// TIA Portal V19 program export: 3 tag tables, 4 data types, 23 data blocks, 30 code blocks (in call order from the OBs), 38 instance data blocks

VAR_GLOBAL   // PLC tag table "Safety_IO"
   IS_EstopLeftRopePull AT %I500.1 : Bool;   // Right e-stop rope pull switch - Channel 1   {ExternalAccessible false}
   IS_EstopRightRopePull AT %I500.0 : Bool;   // Left e-stop rope pull switch - Channel 1   {ExternalAccessible false}
   IS_EStopMainCabinet AT %I500.2 : Bool;   // Main panel e-stop - Channel 1   {ExternalAccessible false}
   IS_EStopEntryDoor AT %I500.3 : Bool;   // Entry door e-stop - Channel 1   {ExternalAccessible false}
   IS_EstopLeftRopePull_Ch2 AT %I500.5 : Bool;   // Right e-stop rope pull switch - Channel 2   {ExternalAccessible false}
   IS_EstopRightRopePull_Ch2 AT %I500.4 : Bool;   // Left e-stop rope pull switch - Channel 2   {ExternalAccessible false}
   IS_EStopMainCabinet_Ch2 AT %I500.6 : Bool;   // Main panel e-stop - Channel 2   {ExternalAccessible false}
   IS_EStopEntryDoor_Ch2 AT %I500.7 : Bool;   // Entry door e-stop - Channel 2   {ExternalAccessible false}
   IS_DoorAcces_Ch1 AT %I507.0 : Bool;   // Door acces state - Channel 1   {ExternalAccessible false}
   IS_GateAccesCBS AT %I507.1 : Bool;   // CBS Gate Acces State - Channel 1   {ExternalAccessible false}
   IS_EStopControlRoom AT %I507.2 : Bool;   // Control Room E-Stop - Channel 1   {ExternalAccessible false}
   IS_DoorAcces_Ch2 AT %I507.4 : Bool;   // Door acces state - Channel 2   {ExternalAccessible false}
   IS_GateAccesCBS_Ch2 AT %I507.5 : Bool;   // CBS Gate Acces State - Channel 2   {ExternalAccessible false}
   IS_EStopControlRoom_Ch2 AT %I507.6 : Bool;   // Control Room E-Stop - Channel 2   {ExternalAccessible false}
   OS_EStopSuctionUnit AT %Q522.1 : Bool;   // E-Stop Suction Unit   {ExternalAccessible false}
   OS_EnableAirSupplyLeftRobot AT %Q522.2 : Bool;   // Air supply robot 1 Ok   {ExternalAccessible false}
   OS_EnableAirSupplyRightRobot AT %Q522.3 : Bool;   // Air supply robot 2 Ok   {ExternalAccessible false}
   OS_EnableAirSupplySuctionUnit AT %Q522.4 : Bool;   // Air supply suction unit Ok   {ExternalAccessible false}
   ISS_EStopSuctionUnit AT %I522.1 : Bool;   // State E-Stop Suction Unit   {ExternalAccessible false}
   ISS_EnableAirSupplyLeftRobot AT %I522.2 : Bool;   // State Air supply robot 1 Ok   {ExternalAccessible false}
   ISS_EnableAirSupplyRightRobot AT %I522.3 : Bool;   // State Air supply robot 2 Ok   {ExternalAccessible false}
   ISS_EnableAirSupplySuctionUnit AT %I522.4 : Bool;   // Air supply suction unit Ok   {ExternalAccessible false}
   ISS_EstopLeftRopePull AT %I501.1 : Bool;   // State Right e-stop rope pull switch - Channel 1   {ExternalAccessible false}
   ISS_EstopRightRopePull AT %I501.0 : Bool;   // State Left e-stop rope pull switch - Channel 1   {ExternalAccessible false}
   ISS_EStopMainCabinet AT %I501.2 : Bool;   // State Main panel e-stop - Channel 1   {ExternalAccessible false}
   ISS_EStopEntryDoor AT %I501.3 : Bool;   // State Entry door e-stop - Channel 1   {ExternalAccessible false}
   ISS_DoorAcces_Ch1 AT %I508.0 : Bool;   // State Door acces state - Channel 1   {ExternalAccessible false}
   ISS_GateAccesCBS AT %I508.1 : Bool;   // State CBS Gate Acces State - Channel 1   {ExternalAccessible false}
   ISS_EStopControlRoom AT %I508.2 : Bool;   // State Control Room E-Stop - Channel 1   {ExternalAccessible false}
   ISS_DoorAcces_Ch2 AT %I508.4 : Bool;   // State Door acces state - Channel 2   {ExternalAccessible false}
   ISB_500 AT %IB500 : SInt;   //    {ExternalWritable false}
   ISB_507 AT %IB507 : SInt;   //    {ExternalWritable false}
   ISB_514 AT %IB514 : SInt;   //    {ExternalWritable false}
   OSB_522 AT %QB522 : SInt;   //    {ExternalWritable false}
   IS_PedestrialDoor AT %I507.3 : Bool;   // Pedestral door acces control   {ExternalAccessible false}
   IS_CaptiveKeyState AT %I514.0 : Bool;   // Captive key in lock - Channel 1   {ExternalAccessible false}
   IS_CaptiveKeyState_Ch2 AT %I514.4 : Bool;   // Captive key in lock - Channel 2   {ExternalAccessible false}
   ISS_CaptiveKeyState AT %I515.0 : Bool;   // State Captive key in lock   {ExternalAccessible false}
   IS_VacuumPumpRunning AT %I507.7 : Bool;   // Vacuum pump runing, zero speed detection   {ExternalAccessible false}
END_VAR

VAR_GLOBAL   // PLC tag table "Standard_IO"
   I_IPBDoorAccesRequest AT %I100.0 : Bool;   // Illuminate push button acces request   {ExternalAccessible false}
   I_IPBCloseDoor AT %I100.1 : Bool;   // Illuminate push button close door   {ExternalAccessible false}
   I_EStopState AT %I100.2 : Bool;   // Entry door AU state   {ExternalAccessible false}
   I_DoorClosed AT %I100.3 : Bool;   // Entry door state 1   {ExternalAccessible false}
   I_BoltTongueInserted AT %I100.4 : Bool;   // Entry door state 2   {ExternalAccessible false}
   I_GuardLocked AT %I100.5 : Bool;   // Entry door state 3   {ExternalAccessible false}
   I_FaultPresent AT %I100.6 : Bool;   // Entry door state 4   {ExternalAccessible false}
   I_PSAirLeftRobotOk AT %I101.0 : Bool;   // Air supply robot 1 Ok   {ExternalAccessible false}
   I_PSAirRightRobotOk AT %I101.1 : Bool;   // Air supply robot 2 Ok   {ExternalAccessible false}
   I_PSAirSuctionUnitOk AT %I101.2 : Bool;   // Air supply suction unit Ok   {ExternalAccessible false}
   I_FanDriveRunning AT %I101.4 : Bool;   // Suction unit - Fan Drive Running   {ExternalAccessible false}
   I_DustBagFull AT %I101.5 : Bool;   // Suction unit - Dust bag full   {ExternalAccessible false}
   I_FanDriveFault AT %I101.6 : Bool;   // Suction unit - Fan Drive fault   {ExternalAccessible false}
   I_SequencerFault AT %I101.7 : Bool;   // Suction unit - Sequencer in fault   {ExternalAccessible false}
   O_IPBDoorAccesRequest AT %Q100.0 : Bool;   // Illuminate push button acces request   {ExternalAccessible false}
   O_IPBCloseDoor AT %Q100.1 : Bool;   // Illuminate push button close door   {ExternalAccessible false}
   O_ResetDoorFault AT %Q100.2 : Bool;   // Reset fault on door   {ExternalAccessible false}
   O_SignalToweGreenLight AT %Q100.4 : Bool;   // Light towers - green light   {ExternalAccessible false}
   O_SignalToweOrangeLight AT %Q100.5 : Bool;   // Light towers - orange light   {ExternalAccessible false}
   O_SignalToweRedLight AT %Q100.6 : Bool;   // Light towers - red light   {ExternalAccessible false}
   O_SignalToweHorn AT %Q100.7 : Bool;   // Light towers - horn   {ExternalAccessible false}
   O_StartVacuum AT %Q101.4 : Bool;   // Suction unit - Vacuum On   {ExternalAccessible false}
   O_StopVacuum AT %Q101.5 : Bool;   // Suction unit - Vacuum Off   {ExternalAccessible false}
   O_TeepTrackCycleTimeR1 AT %Q102.0 : Bool;   // Alstom Teep track Cycle Time Robot 1 (Left)   {ExternalAccessible false}
   O_TeepTrackStartStopR1 AT %Q102.1 : Bool;   // Alstom Teep track Start and Stop Robot 1 (Left)   {ExternalAccessible false}
   O_LockDoor AT %Q101.0 : Bool;   // Lock acces door   {ExternalAccessible false}
   OST_SendLeft AT %Q106.0 : "stMasterToSlave";   // Send information to left slave PLC   {ExternalAccessible false}
   OST_SendRight AT %Q234.0 : "stMasterToSlave";   // Send information to right slave PLC   {ExternalAccessible false}
   IST_ReceiveLeft AT %I106.0 : "stSlaveToMaster";   // Receive information from left slave PLC   {ExternalAccessible false}
   IST_ReceiveRight AT %I234.0 : "stSlaveToMaster";   // Receive information from right slave PLC   {ExternalAccessible false}
   I_FanFault AT %I102.0 : Bool;   // Suction unit - Fan fault   {ExternalAccessible false}
   I_ValveMotorFault AT %I102.1 : Bool;   // Suction unit - Valve Motor Fault   {ExternalAccessible false}
   IB_100 AT %IB100 : SInt;   //    {ExternalWritable false}
   IB_101 AT %IB101 : SInt;   //    {ExternalWritable false}
   IB_102 AT %IB102 : SInt;   //    {ExternalWritable false}
   IB_103 AT %IB103 : SInt;   //    {ExternalWritable false}
   OB_100 AT %QB100 : SInt;   //    {ExternalWritable false}
   OB_101 AT %QB101 : SInt;   //    {ExternalWritable false}
   OB_102 AT %QB102 : SInt;   //    {ExternalWritable false}
   OB_103 AT %QB103 : SInt;   //    {ExternalWritable false}
   O_TeepTrackCycleTimeR2 AT %Q102.2 : Bool;   // Alstom Teep track Cycle Time Robot 2 (Right)   {ExternalAccessible false}
   O_TeepTrackStartStopR2 AT %Q102.3 : Bool;   // Alstom Teep track Start and Stop Robot 2 (Right)   {ExternalAccessible false}
END_VAR

VAR_GLOBAL   // PLC tag table "System"
   System_Byte AT %MB1 : Byte;
   FirstScan AT %M1.0 : Bool;
   DiagStatusUpdate AT %M1.1 : Bool;
   AlwaysTRUE AT %M1.2 : Bool;
   AlwaysFALSE AT %M1.3 : Bool;
   Clock_Byte AT %MB0 : Byte;
   Clock_10Hz AT %M0.0 : Bool;
   Clock_5Hz AT %M0.1 : Bool;
   "Clock_2.5Hz" AT %M0.2 : Bool;
   Clock_2Hz AT %M0.3 : Bool;
   "Clock_1.25Hz" AT %M0.4 : Bool;
   Clock_1Hz AT %M0.5 : Bool;
   "Clock_0.625Hz" AT %M0.6 : Bool;
   "Clock_0.5Hz" AT %M0.7 : Bool;
   ShuntTempSeb AT %M10.0 : Bool;
   ISS_PedestrialDoor AT %I508.3 : Bool;   // State Pedestral door acces control
   ISS_VacuumPumpRunning AT %I508.7 : Bool;   // State Vacuum pump runing, zero speed detection
END_VAR

TYPE "stConfigGrease"
   STRUCT
      uiNbPulsePerKm : UInt := 4411;   // Number of pulse per km
      uiKmForGreasing : UInt := 32;   // Number of Km between each greasing
      tTimeEnableGreasePump : Time := T#1M;   // Time of enabling grease pump
      tTimeoutPxGrease : Time := T#1M;   // Timeout for the proxy greas
   END_STRUCT;
END_TYPE

TYPE "stFlatnessData"
   STRUCT
      xFlatnessCrtlRequestRecord { ExternalAccessible := 'False'; ExternalVisible := 'False'; ExternalWritable := 'False'} : Bool;
      xFlatnessCtrlRecorded { ExternalAccessible := 'False'; ExternalVisible := 'False'; ExternalWritable := 'False'} : Bool;
      xFlatnessCtrlPassed { ExternalAccessible := 'False'; ExternalVisible := 'False'; ExternalWritable := 'False'} : Bool;
      uiStrokePositionDiskA { ExternalAccessible := 'False'; ExternalVisible := 'False'; ExternalWritable := 'False'} : UInt;
      uiStrokePositionDiskB { ExternalAccessible := 'False'; ExternalVisible := 'False'; ExternalWritable := 'False'} : UInt;
      uiStrokePositionDiskC { ExternalAccessible := 'False'; ExternalVisible := 'False'; ExternalWritable := 'False'} : UInt;
   END_STRUCT;
END_TYPE

TYPE "stItemListRecipe"
   STRUCT
      RecipeName { ExternalAccessible := 'False'; ExternalVisible := 'False'; ExternalWritable := 'False'} : String[30];
      RecipeIndex { ExternalAccessible := 'False'; ExternalVisible := 'False'; ExternalWritable := 'False'} : USInt;
   END_STRUCT;
END_TYPE

TYPE "stParamManuFerRobotic"
   STRUCT
      "#OutToSlave.ManualSandingPaperParam.nSetForceTarget    #OutToSlave.ManualSandingPaperParam.nSetForceZero    #OutToSlave.ManualSa" : Bool;
   END_STRUCT;
END_TYPE

DATA_BLOCK "DB_CurrentRecipe"   // DB5
{ S7_Optimized_Access := 'TRUE'; DB_Accessible_From_OPC_UA := 'FALSE' }
// stored: AutoNumber false, DBAccessibleFromOPCUA false, DBAccessibleFromWebserver false, MemoryReserve 100
   VAR RETAIN
      usiCurrentRecipeNumber : USInt;
      usiCurrentLayerType : USInt;
      usiCurrentJobDataLeft { ExternalAccessible := 'False'; ExternalVisible := 'False'; ExternalWritable := 'False'} : USInt;
      usiCurrentJobDataRight { ExternalAccessible := 'False'; ExternalVisible := 'False'; ExternalWritable := 'False'} : USInt;
      uiCdbNumber : UInt;
      CompleteRecipe : "stRecipe";
      WorkRecipe { S7_SetPoint := 'True'} : "stWorkRecipe";
   END_VAR
BEGIN
END_DATA_BLOCK

DATA_BLOCK "DB_Exchange"   // DB1
{ S7_Optimized_Access := 'TRUE'; DB_Accessible_From_OPC_UA := 'FALSE' }
// stored: AutoNumber false, DBAccessibleFromOPCUA false, DBAccessibleFromWebserver false, MemoryReserve 100
   VAR
      xAutoMode { ExternalAccessible := 'False'; ExternalVisible := 'False'; ExternalWritable := 'False'} : Bool;   // Automatic mode
      xSemiAutoMode { ExternalAccessible := 'False'; ExternalVisible := 'False'; ExternalWritable := 'False'} : Bool;   // Semi-automatic mode
      xMaintenanceMode { ExternalAccessible := 'False'; ExternalVisible := 'False'; ExternalWritable := 'False'} : Bool;   // Maintenance mode
      xAuthorizationStartSanding { ExternalAccessible := 'False'; ExternalVisible := 'False'; ExternalWritable := 'False'} : Bool;
      xLeftRobotStartVacuum { ExternalAccessible := 'False'; ExternalVisible := 'False'; ExternalWritable := 'False'} : Bool;   // Left Robot request start vacuum
      xRightRobotStartVacuum { ExternalAccessible := 'False'; ExternalVisible := 'False'; ExternalWritable := 'False'} : Bool;   // Right Robot request start vacuum
      xStopRobotRequested { ExternalAccessible := 'False'; ExternalVisible := 'False'; ExternalWritable := 'False'} : Bool;   // Stop robot requested for openning the door
      xLeftRobotStopped { ExternalAccessible := 'False'; ExternalVisible := 'False'; ExternalWritable := 'False'} : Bool;   // Left Robot stopped in good position
      xRightRobotStopped { ExternalAccessible := 'False'; ExternalVisible := 'False'; ExternalWritable := 'False'} : Bool;   // Right Robot stopped in good position
      xGlobalFault { ExternalAccessible := 'False'; ExternalVisible := 'False'; ExternalWritable := 'False'} : Bool;   // Cell Global Fault
      xGlobalWarning { ExternalAccessible := 'False'; ExternalVisible := 'False'; ExternalWritable := 'False'} : Bool;   // Cell Global warning
      xInformation { ExternalAccessible := 'False'; ExternalVisible := 'False'; ExternalWritable := 'False'} : Bool;   // An information message is display
      xConditionOk { ExternalAccessible := 'False'; ExternalVisible := 'False'; ExternalWritable := 'False'} : Bool;   // Condition to run ok
      xStartUpWarningLeft { ExternalAccessible := 'False'; ExternalVisible := 'False'; ExternalWritable := 'False'} : Bool;   // Start up warning before left robot run
      xStartUpWarningRight { ExternalAccessible := 'False'; ExternalVisible := 'False'; ExternalWritable := 'False'} : Bool;   // Start up warning before right robot run
      xReqOperatorAction { ExternalAccessible := 'False'; ExternalVisible := 'False'; ExternalWritable := 'False'} : Bool;   // Request operator action
      xRecipeOpeInProgress { ExternalAccessible := 'False'; ExternalVisible := 'False'; ExternalWritable := 'False'} : Bool;   // Recipe Operation in progress
      xSandingInProgress { ExternalAccessible := 'False'; ExternalVisible := 'False'; ExternalWritable := 'False'} : Bool;   // Sanding process is in progress
      xUnloadRecipe { ExternalAccessible := 'False'; ExternalVisible := 'False'; ExternalWritable := 'False'} : Bool;   // Unload current recipe
      xProductionRunningRobot1 { ExternalAccessible := 'False'; ExternalVisible := 'False'; ExternalWritable := 'False'} : Bool;   // Production running on Robot 1
      xProductionRunningRobot2 { ExternalAccessible := 'False'; ExternalVisible := 'False'; ExternalWritable := 'False'} : Bool;   // Production running on Robot 2
      xStartSanding { ExternalAccessible := 'False'; ExternalVisible := 'False'; ExternalWritable := 'False'} : Bool;   // Beginning of sanding
      xEndSanding { ExternalAccessible := 'False'; ExternalVisible := 'False'; ExternalWritable := 'False'} : Bool;   // End of sanding
      udiVacuumRunningTime { ExternalAccessible := 'False'; ExternalVisible := 'False'; ExternalWritable := 'False'} : UDInt;   // Vacuum Running time
      LeftRobot { ExternalAccessible := 'False'; ExternalVisible := 'False'; ExternalWritable := 'False'} : Struct
         udiFaultTime : UDInt;
         udiRunTime : UDInt;
         udiPauseTime : UDInt;
         udiRobotPowerOnTime : UDInt;
         udiRobotDriveOnTime : UDInt;
         xRobotUsed : Bool;
      END_STRUCT;
      RightRobot { ExternalAccessible := 'False'; ExternalVisible := 'False'; ExternalWritable := 'False'} : Struct
         udiFaultTime : UDInt;
         udiRunTime : UDInt;
         udiPauseTime : UDInt;
         udiRobotPowerOnTime : UDInt;
         udiRobotDriveOnTime : UDInt;
         xRobotUsed : Bool;
      END_STRUCT;
      stLeftRobotFlatnessCtrlData { ExternalAccessible := 'False'; ExternalVisible := 'False'; ExternalWritable := 'False'} : "stFlatnessData";
      stRightRobotFlatnessCtrlData { ExternalAccessible := 'False'; ExternalVisible := 'False'; ExternalWritable := 'False'} : "stFlatnessData";
   END_VAR
BEGIN
END_DATA_BLOCK

DATA_BLOCK "DB_JobData"   // DB3
{ S7_Optimized_Access := 'TRUE'; DB_Accessible_From_OPC_UA := 'FALSE' }
// stored: AutoNumber false, DBAccessibleFromOPCUA false, DBAccessibleFromWebserver false, MemoryReserve 100
   VAR RETAIN
      aJobData : Array[0..99] of "stJobData";   // Array of job data parameters
   END_VAR
BEGIN
END_DATA_BLOCK

DATA_BLOCK "DB_Parameters"   // DB2
{ S7_Optimized_Access := 'TRUE'; DB_Accessible_From_OPC_UA := 'FALSE' }
// stored: DBAccessibleFromOPCUA false, DBAccessibleFromWebserver false, MemoryReserve 100
   VAR RETAIN
      CommMainPanel { ExternalAccessible := 'False'; ExternalVisible := 'False'; ExternalWritable := 'False'} : TCON_IP_v4;
      CommLeftRobot { ExternalAccessible := 'False'; ExternalVisible := 'False'; ExternalWritable := 'False'} : TCON_IP_v4;
      CommRightRobot { ExternalAccessible := 'False'; ExternalVisible := 'False'; ExternalWritable := 'False'} : TCON_IP_v4;
      tDelatBetweenReady { ExternalAccessible := 'False'; ExternalVisible := 'False'; ExternalWritable := 'False'} : Time := T#1s;
   END_VAR
BEGIN
   CommMainPanel.InterfaceId := 64;
   CommMainPanel.ID := 16#01;
   CommMainPanel.ConnectionType := 16#0B;
   CommMainPanel.ActiveEstablished := TRUE;
   CommMainPanel.RemoteAddress.ADDR[1] := 192;
   CommMainPanel.RemoteAddress.ADDR[2] := 168;
   CommMainPanel.RemoteAddress.ADDR[3] := 1;
   CommMainPanel.RemoteAddress.ADDR[4] := 20;
   CommMainPanel.RemotePort := 502;
   CommLeftRobot.InterfaceId := 64;
   CommLeftRobot.ID := 16#02;
   CommLeftRobot.ConnectionType := 16#0B;
   CommLeftRobot.ActiveEstablished := TRUE;
   CommLeftRobot.RemoteAddress.ADDR[1] := 192;
   CommLeftRobot.RemoteAddress.ADDR[2] := 168;
   CommLeftRobot.RemoteAddress.ADDR[3] := 1;
   CommLeftRobot.RemoteAddress.ADDR[4] := 21;
   CommLeftRobot.RemotePort := 502;
   CommRightRobot.InterfaceId := 64;
   CommRightRobot.ID := 16#03;
   CommRightRobot.ConnectionType := 16#0B;
   CommRightRobot.ActiveEstablished := TRUE;
   CommRightRobot.RemoteAddress.ADDR[1] := 192;
   CommRightRobot.RemoteAddress.ADDR[2] := 168;
   CommRightRobot.RemoteAddress.ADDR[3] := 1;
   CommRightRobot.RemoteAddress.ADDR[4] := 22;
   CommRightRobot.RemotePort := 503;
END_DATA_BLOCK

DATA_BLOCK "DB_FromHmi"   // DB29
{ S7_Optimized_Access := 'TRUE'; DB_Accessible_From_OPC_UA := 'FALSE' }
// stored: AutoNumber false, DBAccessibleFromOPCUA false, DBAccessibleFromWebserver false, MemoryReserve 100
   VAR
      xLightTest : Bool;   // Light test
      xResetFault : Bool;   // Reset fault and safety
      xStartVacuum : Bool;   // Start vacuum
      xStopVacuum : Bool;   // Stop vacuum
      xReqChangeBigbag : Bool;   // Request change Bigbag
      xValidationBigbagChanged : Bool;   // Validation operator bigbag changed
      xListRecipe : Bool;   // Do the list of all the recipe available in the data base
      xLoadRecipe : Bool;   // Load current recipe from data base
      xSaveRecipe : Bool;   // Save current recipe into the data base
      xNewRecipe : Bool;   // Select next free recipe on the data base
      xDeleteRecipe : Bool;   // Delete the recipe from the data base
      xNextRecipe : Bool;   // Load next recipe in the data base
      xPrevRecipe : Bool;   // Load previus recipe in the data base
      xValideOperation : Bool;   // Validation Operator to remove or Put disk on FerRobotic head
      xValideFault : Bool;   // Validation Operator of Flatness fault
      xProdRecordNext : Bool;
      xProdRecordPrev : Bool;
      xProdRecordDeleteAll : Bool;
      xFlatRecNextLeftRobot : Bool;
      xFlatRecPrevLeftRobot : Bool;
      xFlatRecDelAllLeftRobot : Bool;
      xFlatRecNextRightRobot : Bool;
      xFlatRecPrevRightRobot : Bool;
      xFlatRecDelAllRightRobot : Bool;
   END_VAR
   VAR RETAIN
      xEnableStartLeftRobot : Bool;   // Enable start robot
      xEnableStartRightRobot : Bool;   // Enable start robot
   END_VAR
   VAR
      xDryRun : Bool;   // Robot run in DryRun
      xExportProdData : Bool;
      xExportFlatCtrlRobot1 : Bool;
      xExportFlatCtrlRobot2 : Bool;
      uiCurentRecord : UInt;
      uiFlatCurentRecLeftRobot : UInt;
      uiFlatCurentRecRightRobot : UInt;
      uiDisplayJobNumber : UInt;
   END_VAR
   VAR RETAIN
      usiOperatingMode : USInt;   // Operating mode (1 = Semi-Auto, 2 = Auto)
      uiUserGroup : USInt;   // User grope number logged on HMI
   END_VAR
   VAR
      LeftRobot : Struct   // Command for left robot
         xResetGrafcet : Bool;   // Reset robot communication grafcet
         xStartCycle : Bool;   // Start Cycle
         xStopCycle : Bool;   // Stop Cycle
         xCancelCycle : Bool;   // Cancel cycle
         xStopEndCycle : Bool;   // Stop end of cycle
         xReqChangeDisk : Bool;
         xStartServicePath : Bool;   // Start service path
         xStopServicePath : Bool;   // Stop service path
         xCancelServicePath : Bool;   // Cancel service path
         usiJobNumberDisplay : USInt;   // Job number displayed for robot left
         uiServicePathNumber : UInt;   // Service path number
         xCmdManuLockGimball : Bool;
         xCmdManuLockEccentric1 : Bool;
         xCmdManuLockEccentric2 : Bool;
         xCmdManuLockEccentric3 : Bool;
         xCmdManuEnableRotate : Bool;
         xCmdManuCloseVacValve : Bool;
         xCmdManuOpenVacValve : Bool;
         xCmdManuRemoveConfig : Bool;   // Manual command for activate the Remove config on FerRobotic Head
         xCmdManuPickupConfig : Bool;   // Manual command for activate the Pickup config on FerRobotic Head
         xCmdManuFlatnessConfig : Bool;   // Manual command for activate the Flatness check config on FerRobotic Head
         xMaintStartProg : Bool;
         xMaintStartMain : Bool;
         xForceLubricationX : Bool;
         xForceLubricationZ : Bool;
         ParamManu : "stFerRoboticParam";
      END_STRUCT;
      RightRobot : Struct   // Commande for right robot
         xResetGrafcet : Bool;   // Reset robot communication grafcet
         xStartCycle : Bool;   // Start Cycle
         xStopCycle : Bool;   // Stop Cycle
         xCancelCycle : Bool;   // Cancel cycle
         xStopEndCycle : Bool;   // Stop end of cycle
         xReqChangeDisk : Bool;
         xStartServicePath : Bool;   // Start service path
         xStopServicePath : Bool;   // Stop service path
         xCancelServicePath : Bool;   // Cancel service path
         usiJobNumberDisplay : USInt;   // Job number displayed for robot right
         uiServicePathNumber : UInt;   // Service path number
         xCmdManuLockGimball : Bool;
         xCmdManuLockEccentric1 : Bool;
         xCmdManuLockEccentric2 : Bool;
         xCmdManuLockEccentric3 : Bool;
         xCmdManuEnableRotate : Bool;
         xCmdManuCloseVacValve : Bool;
         xCmdManuOpenVacValve : Bool;
         xCmdManuRemoveConfig : Bool;   // Manual command for activate the Remove config on FerRobotic Head
         xCmdManuPickupConfig : Bool;   // Manual command for activate the Pickup config on FerRobotic Head
         xCmdManuFlatnessConfig : Bool;   // Manual command for activate the Flatness check config on FerRobotic Head
         xMaintStartProg : Bool;
         xMaintStartMain : Bool;
         xForceLubricationX : Bool;
         xForceLubricationZ : Bool;
         ParamManu : "stFerRoboticParam";
      END_STRUCT;
   END_VAR
BEGIN
END_DATA_BLOCK

DATA_BLOCK "DB_HmiLight"   // DB27
{ S7_Optimized_Access := 'TRUE' }
// stored: AutoNumber false, MemoryReserve 100
   VAR
      xMemFpClock { ExternalAccessible := 'False'; ExternalVisible := 'False'; ExternalWritable := 'False'} : Bool;
      xFpClock { ExternalAccessible := 'False'; ExternalVisible := 'False'; ExternalWritable := 'False'} : Bool;
   END_VAR
BEGIN
END_DATA_BLOCK

DATA_BLOCK "DB_PointerHMI"   // DB25
{ S7_Optimized_Access := 'TRUE'; DB_Accessible_From_OPC_UA := 'FALSE' }
// stored: AutoNumber false, DBAccessibleFromOPCUA false, DBAccessibleFromWebserver false, MemoryReserve 100
   VAR
      Coordination : Word;
      ProjectID : Word;
      ScreenNumber : Array[0..4] of Word;
      JobMailbox : Array[0..3] of Word;
   END_VAR
BEGIN
END_DATA_BLOCK

DATA_BLOCK "DB_ToHmi"   // DB28
{ S7_Optimized_Access := 'TRUE'; DB_Accessible_From_OPC_UA := 'FALSE' }
// stored: AutoNumber false, DBAccessibleFromOPCUA false, DBAccessibleFromWebserver false, MemoryReserve 100
   VAR
      xShowPopReqChangeBigbag : Bool;   // Show Popup change Bigbag requested
      xShowPopNoMoreRecipeAvailable : Bool;   // Show Popup no more recipe available in the data base
      xSafetyState { ExternalWritable := 'False'} : Bool;   // Safety State
      xDiseableRecipeButton { ExternalWritable := 'False'} : Bool;   // Diseable all button for manage recipe
      xDisplayPrevButton { ExternalWritable := 'False'} : Bool;   // Display previous button in recipe screen
      xDisplayNextButton { ExternalWritable := 'False'} : Bool;   // Display next button in recipe screen
      xDiseableNewButton { ExternalWritable := 'False'} : Bool;   // Diseable new recipe button
      xDiseableSaveButton { ExternalWritable := 'False'} : Bool;   // Diseable save recipe button
      xDiseableDeleteButton { ExternalWritable := 'False'} : Bool;   // Diseable delete recipe button
      xLockRecipe { ExternalWritable := 'False'} : Bool;   // Lock recipe during production
      xLockSelectJobDataNumber { ExternalWritable := 'False'} : Bool;   // Lock selection of job data number
      xLockJobDataLeft { ExternalWritable := 'False'} : Bool;   // Lock modification Job Data left robot
      xLockJobDataRight { ExternalWritable := 'False'} : Bool;   // Lock modification Job Data right robot
      xVacuumPumpRunning { ExternalWritable := 'False'} : Bool;
      xVacuumDriveActivated { ExternalWritable := 'False'} : Bool;
      xLockMaintenance { ExternalWritable := 'False'} : Bool;   // Lock button to switch in Maintenance mode
      xLockSemiAuto { ExternalWritable := 'False'} : Bool;   // Lock button to switch in Semi-Auto mode
      xHomePositionR1 { ExternalWritable := 'False'} : Bool;   // Robot 1 in Home Position
      xHomePositionR2 { ExternalWritable := 'False'} : Bool;   // Robot 2 in Home Position
      xAccessDoor { ExternalWritable := 'False'} : Bool;   // Access door closed
      xCaptiveKey { ExternalWritable := 'False'} : Bool;   // Captive key on contact switch
      xLightBeam { ExternalWritable := 'False'} : Bool;   // Light Beam clear
      xCbsGate { ExternalWritable := 'False'} : Bool;   // CBS Gate closed
      nGlobalState { ExternalWritable := 'False'} : Int;   // Cell global state
      wVacuumState { ExternalWritable := 'False'} : Word;
      uiProdRecordMin { ExternalWritable := 'False'} : UInt;   // Mini record number
      uiProdRecordMax { ExternalWritable := 'False'} : UInt;   // Maxi record number
      uiFlatRecMinLeftRobot { ExternalWritable := 'False'} : UInt;   // Mini record number for Flatness Left robot
      uiFlatRecMaxLeftRobot { ExternalWritable := 'False'} : UInt;   // Maxi record number for Flatness Left robot
      uiFlatRecMinRightRobot { ExternalWritable := 'False'} : UInt;   // Mini record number for Flatness Right robot
      uiFlatRecMaxRightRobot { ExternalWritable := 'False'} : UInt;   // Maxi record number for Flatness Right robot
      uiNbrDisplyedLine { ExternalWritable := 'False'} : UInt;   // Number of displayed lime of production
      uiFirstRecordDisplayed { ExternalWritable := 'False'} : UInt;   // First record displayed
      uiLastRecordDisplayed { ExternalWritable := 'False'} : UInt;   // Last record displayed
      sVacuumRunningTime { ExternalWritable := 'False'} : String[15];
      LeftRobot : Struct
         xRobotInAuto { ExternalWritable := 'False'} : Bool;
         xRobotInManu { ExternalWritable := 'False'} : Bool;
         xRobotReqReset { ExternalWritable := 'False'} : Bool;
         xRecipeInProgress { ExternalWritable := 'False'} : Bool;
         xPathInProgress { ExternalWritable := 'False'} : Bool;   // Service path in progress
         xPathStopped { ExternalWritable := 'False'} : Bool;   // Service path stopped
         xPathCancelled { ExternalWritable := 'False'} : Bool;   // Service path cancelled
         xContactState { ExternalWritable := 'False'} : Bool;   // State of the FerRobotic head contact
         xShowPopRemoveDisk : Bool;
         xShowPopPickupDisk : Bool;
         xShowPopFlatnessFault : Bool;
         xMagazineEmpty { ExternalWritable := 'False'} : Bool;
         xRangeFinderDetection { ExternalWritable := 'False'} : Bool;
         xValveOpen { ExternalWritable := 'False'} : Bool;
         xValveClosed { ExternalWritable := 'False'} : Bool;
         uiRangeFinderValue { ExternalWritable := 'False'} : UInt;
         nActualForce { ExternalWritable := 'False'} : Int;   // Actual force on FerRobotic head
         rActualPosition { ExternalWritable := 'False'} : Real;   // Actual position of the FerRobotic head
         uiActualJobDataNumber { ExternalWritable := 'False'} : UInt;
         uiNbDiskUsed { ExternalWritable := 'False'} : UInt;
         uiRobotStatus { ExternalWritable := 'False'} : UInt;
         uiSetSpeed { ExternalWritable := 'False'} : UInt;
         uiRobotSpeed { ExternalWritable := 'False'} : UInt;
         uiPaperChangeDistance { ExternalWritable := 'False'} : UInt;
         uiCounterPulse_X { ExternalWritable := 'False'} : UInt;
         uiCounterPulse_Z { ExternalWritable := 'False'} : UInt;
         uiGreaseFault_X { ExternalWritable := 'False'} : UInt;
         uiGreaseFault_Z { ExternalWritable := 'False'} : UInt;
         uiDistanceSandingDisk { ExternalWritable := 'False'} : UInt;
         uiActualRobotSpeed { ExternalWritable := 'False'} : UInt;   // Actual speed of theTCP of the robot
         uiDistanceBeforeGreasingX : UInt;
         uiDistanceBeforeGreasingZ : UInt;
         udiOdometer_X { ExternalWritable := 'False'} : UDInt;
         udiOdometer_Z { ExternalWritable := 'False'} : UDInt;
         sRunTime { ExternalWritable := 'False'} : String[12];
         sPauseTime { ExternalWritable := 'False'} : String[12];
         sFaultTime { ExternalWritable := 'False'} : String[12];
         sRobotPowerOnTime { ExternalWritable := 'False'} : String[15];
         sRobotDriveOnTime { ExternalWritable := 'False'} : String[15];
         IB_Safety500 { ExternalWritable := 'False'} : SInt;
         IB_Input100 { ExternalWritable := 'False'} : SInt;
         IB_Input101 { ExternalWritable := 'False'} : SInt;
         IB_Input102 { ExternalWritable := 'False'} : SInt;
         IB_Input103 { ExternalWritable := 'False'} : SInt;
         IN_Input600 { ExternalWritable := 'False'} : Int;
         IN_Input602 { ExternalWritable := 'False'} : Int;
         IN_Input604 { ExternalWritable := 'False'} : Int;
         IN_Input606 { ExternalWritable := 'False'} : Int;
         OB_Safety508 { ExternalWritable := 'False'} : SInt;
         OB_Output100 { ExternalWritable := 'False'} : SInt;
         OB_Output101 { ExternalWritable := 'False'} : SInt;
         IB_Fast90 { ExternalWritable := 'False'} : SInt;
      END_STRUCT;
      RightRobot : Struct
         xRobotInAuto { ExternalWritable := 'False'} : Bool;
         xRobotInManu { ExternalWritable := 'False'} : Bool;
         xRobotReqReset { ExternalWritable := 'False'} : Bool;
         xRecipeInProgress { ExternalWritable := 'False'} : Bool;
         xPathInProgress { ExternalWritable := 'False'} : Bool;   // Service path in progress
         xPathStopped { ExternalWritable := 'False'} : Bool;   // Service path stopped
         xPathCancelled { ExternalWritable := 'False'} : Bool;   // Service path cancelled
         xContactState { ExternalWritable := 'False'} : Bool;   // State of the FerRobotic head contact
         xShowPopRemoveDisk : Bool;
         xShowPopPickupDisk : Bool;
         xShowPopFlatnessFault : Bool;
         xMagazineEmpty { ExternalWritable := 'False'} : Bool;
         xRangeFinderDetection { ExternalWritable := 'False'} : Bool;
         xValveOpen { ExternalWritable := 'False'} : Bool;
         xValveClosed { ExternalWritable := 'False'} : Bool;
         uiRangeFinderValue { ExternalWritable := 'False'} : UInt;
         nActualForce { ExternalWritable := 'False'} : Int;   // Actual force on FerRobotic head
         rActualPosition { ExternalWritable := 'False'} : Real;   // Actual position of the FerRobotic head
         uiActualJobDataNumber { ExternalWritable := 'False'} : UInt;
         uiNbDiskUsed { ExternalWritable := 'False'} : UInt;
         uiRobotStatus { ExternalWritable := 'False'} : UInt;
         uiSetSpeed { ExternalWritable := 'False'} : UInt;
         uiRobotSpeed { ExternalWritable := 'False'} : UInt;
         uiPaperChangeDistance { ExternalWritable := 'False'} : UInt;
         uiCounterPulse_X { ExternalWritable := 'False'} : UInt;
         uiCounterPulse_Z { ExternalWritable := 'False'} : UInt;
         uiGreaseFault_X { ExternalWritable := 'False'} : UInt;
         uiGreaseFault_Z { ExternalWritable := 'False'} : UInt;
         uiDistanceSandingDisk { ExternalWritable := 'False'} : UInt;
         uiActualRobotSpeed { ExternalWritable := 'False'} : UInt;   // Actual speed of theTCP of the robot
         uiDistanceBeforeGreasingX : UInt;
         uiDistanceBeforeGreasingZ : UInt;
         udiOdometer_X { ExternalWritable := 'False'} : UDInt;
         udiOdometer_Z { ExternalWritable := 'False'} : UDInt;
         sRunTime { ExternalWritable := 'False'} : String[12];
         sPauseTime { ExternalWritable := 'False'} : String[12];
         sFaultTime { ExternalWritable := 'False'} : String[12];
         sRobotPowerOnTime { ExternalWritable := 'False'} : String[15];
         sRobotDriveOnTime { ExternalWritable := 'False'} : String[15];
         IB_Safety500 { ExternalWritable := 'False'} : SInt;
         IB_Input100 { ExternalWritable := 'False'} : SInt;
         IB_Input101 { ExternalWritable := 'False'} : SInt;
         IB_Input102 { ExternalWritable := 'False'} : SInt;
         IB_Input103 { ExternalWritable := 'False'} : SInt;
         IN_Input600 { ExternalWritable := 'False'} : Int;
         IN_Input602 { ExternalWritable := 'False'} : Int;
         IN_Input604 { ExternalWritable := 'False'} : Int;
         IN_Input606 { ExternalWritable := 'False'} : Int;
         OB_Safety508 { ExternalWritable := 'False'} : SInt;
         OB_Output100 { ExternalWritable := 'False'} : SInt;
         OB_Output101 { ExternalWritable := 'False'} : SInt;
         IB_Fast90 { ExternalWritable := 'False'} : SInt;
      END_STRUCT;
      aRecipeList { ExternalWritable := 'False'} : Array[1..10] of "stRecipeListHMI";   // List of the recipe name display on HMI
      DataSentronMainPanel { ExternalWritable := 'False'} : "Sentron_PAC";   // Sentron main panel data
      DateSentronLeftRobot { ExternalWritable := 'False'} : "Sentron_PAC";   // Sentron left robot data
      DataSentronRightRobot { ExternalWritable := 'False'} : "Sentron_PAC";   // Sentron right robot data
      Fault { ExternalWritable := 'False'} : Struct
         wFerRoboticLeft : Word;
         wManageRobotLeft : Word;
         wOtherLeft : Word;
         wRobotLeft : Word;
         wVacuumValveLeft : Word;
         wFerRoboticManageLeft : Word;
         wFault07 : Word;
         wFault08 : Word;
         wFerRoboticRight : Word;
         wManageRobotRight : Word;
         wOtherRight : Word;
         wRobotRight : Word;
         wVacuumValveRight : Word;
         wFerRoboticManageRight : Word;
         wFault11 : Word;
         wFault12 : Word;
         wSafetFault : Word;
         wVacuumFault : Word;
         wSafetyModule : Word;
         wOtherMaster : Word;
         wFault15 : Word;
         wFault16 : Word;
         wFault17 : Word;
         wFault18 : Word;
      END_STRUCT;
      Warning { ExternalWritable := 'False'} : Struct
         wSafetyComp : Word;
         wWarnigLeft : Word;
         wWarnigRight : Word;
         wWarnig04 : Word;
         wWarnig05 : Word;
         wWarnig06 : Word;
         wWarnig07 : Word;
         wWarnig08 : Word;
         wWarnig09 : Word;
         wWarnig10 : Word;
      END_STRUCT;
      Message { ExternalWritable := 'False'} : Struct
         wMessage01 : Word;
         wMessage02 : Word;
         wMessage03 : Word;
         wMessage04 : Word;
      END_STRUCT;
      aDisplayProdData { ExternalWritable := 'False'} : Array[0..9] of "stProductionRecord";
      DisplayFlatRecLeftRobot { ExternalWritable := 'False'} : "stFlatnessCtrlRecord";
      DisplayFlatRecRightRobot { ExternalWritable := 'False'} : "stFlatnessCtrlRecord";
   END_VAR
BEGIN
END_DATA_BLOCK

DATA_BLOCK "DB_SNTP_Diag"   // DB202
{ S7_Optimized_Access := 'TRUE' }
// stored: AutoNumber false, MemoryReserve 100
   VAR
      error : Bool;   // An error occured
      statusID : Int;   // Specifies the source of the error (1 = TCON, 2 = TUSEND, 3 = TURCV)
      status : Word;   // Specifies the error
      lastStatusID : Int;   // Saved status ID
      lastStatus : Word;   // Saved status
   END_VAR
BEGIN
END_DATA_BLOCK

DATA_BLOCK "DB_SNTP_Param"   // DB201
{ S7_Optimized_Access := 'TRUE' }
// stored: AutoNumber false, MemoryReserve 100
   VAR
      referenceID : USInt;   // Source of date and time (0 = uncalibrated local clock, 1 = DCF77, 2 = GPS)
      lastTimeSet : DTL := DTL#1990-01-01-00:00:00;   // Date and time when the time was set last. Set only if external reference is used.
      connID : CONN_OUC := 16#0FFF;   // Internal connection ID used for TURCV and TUSEND
   END_VAR
BEGIN
END_DATA_BLOCK

DATA_BLOCK "DB_CommSlave"   // DB40
{ S7_Optimized_Access := 'TRUE' }
// stored: AutoNumber false, MemoryReserve 100
   VAR
      Left { ExternalAccessible := 'False'; ExternalVisible := 'False'; ExternalWritable := 'False'} : Struct
         xRobotHasStarted : Bool;   // Robot has started
         xRobotHasFinished : Bool;   // Robot has finished
         xBothSideFinished : Bool;   // Both robot finished
      END_STRUCT;
      Right { ExternalAccessible := 'False'; ExternalVisible := 'False'; ExternalWritable := 'False'} : Struct
         xRobotHasStarted : Bool;   // Robot has started
         xRobotHasFinished : Bool;   // Robot has finished
         xBothSideFinished : Bool;   // Both robot finished
      END_STRUCT;
   END_VAR
BEGIN
END_DATA_BLOCK

DATA_BLOCK "DB_RecipeEmpty"   // DB51
{ S7_Optimized_Access := 'TRUE' }
// stored: AutoNumber false, MemoryReserve 100
   VAR
      RecipeEmpty { ExternalAccessible := 'False'; ExternalVisible := 'False'; ExternalWritable := 'False'} : "stRecipe";
   END_VAR
BEGIN
   RecipeEmpty.RecipeLayerType[1].RecipeLayerTypeName := 'Putty';
   RecipeEmpty.RecipeLayerType[1].JobTableLeft[0].SetForceZero := 0;
   RecipeEmpty.RecipeLayerType[2].JobTableLeft[0].SetForceZero := 0;
   RecipeEmpty.RecipeLayerType[1].JobTableLeft[0].SetForceTarget := 0;
   RecipeEmpty.RecipeLayerType[2].JobTableLeft[0].SetForceTarget := 0;
   RecipeEmpty.RecipeLayerType[1].JobTableLeft[0].SetTimeRamp := 0;
   RecipeEmpty.RecipeLayerType[2].JobTableLeft[0].SetTimeRamp := 0;
   RecipeEmpty.RecipeLayerType[1].JobTableLeft[0].SetSpeed := 0;
   RecipeEmpty.RecipeLayerType[2].JobTableLeft[0].SetSpeed := 0;
   RecipeEmpty.RecipeLayerType[1].JobTableLeft[0].SetRobotSpeed := 0;
   RecipeEmpty.RecipeLayerType[2].JobTableLeft[0].SetRobotSpeed := 0;
   RecipeEmpty.RecipeLayerType[1].JobTableLeft[0].WornPaperDistance := 0;
   RecipeEmpty.RecipeLayerType[2].JobTableLeft[0].WornPaperDistance := 0;
   RecipeEmpty.RecipeLayerType[1].JobTableLeft[0].Gimball := 0;
   RecipeEmpty.RecipeLayerType[2].JobTableLeft[0].Gimball := 0;
   RecipeEmpty.RecipeLayerType[1].JobTableRight[0].SetForceZero := 0;
   RecipeEmpty.RecipeLayerType[2].JobTableRight[0].SetForceZero := 0;
   RecipeEmpty.RecipeLayerType[1].JobTableRight[0].SetForceTarget := 0;
   RecipeEmpty.RecipeLayerType[2].JobTableRight[0].SetForceTarget := 0;
   RecipeEmpty.RecipeLayerType[1].JobTableRight[0].SetTimeRamp := 0;
   RecipeEmpty.RecipeLayerType[2].JobTableRight[0].SetTimeRamp := 0;
   RecipeEmpty.RecipeLayerType[1].JobTableRight[0].SetSpeed := 0;
   RecipeEmpty.RecipeLayerType[2].JobTableRight[0].SetSpeed := 0;
   RecipeEmpty.RecipeLayerType[1].JobTableRight[0].SetRobotSpeed := 0;
   RecipeEmpty.RecipeLayerType[2].JobTableRight[0].SetRobotSpeed := 0;
   RecipeEmpty.RecipeLayerType[1].JobTableRight[0].WornPaperDistance := 0;
   RecipeEmpty.RecipeLayerType[2].JobTableRight[0].WornPaperDistance := 0;
   RecipeEmpty.RecipeLayerType[1].JobTableRight[0].Gimball := 0;
   RecipeEmpty.RecipeLayerType[2].JobTableRight[0].Gimball := 0;
END_DATA_BLOCK

DATA_BLOCK "DB_Recipes"   // DB50
{ S7_Optimized_Access := 'TRUE' }
// stored: AutoNumber false, IsOnlyStoredInLoadMemory true, MemoryReserve 100
   VAR RETAIN
      aRecipe : Array[0..256] of "stRecipe";
   END_VAR
BEGIN
   aRecipe[1].RecipeName := 'Test Flate Plate';
   aRecipe[2].RecipeName := 'Test Carbody Shell';
   aRecipe[3].RecipeName := 'RGCC5';
   aRecipe[4..23].RecipeName := '';
   aRecipe[1].RecipeCbsType := 'Flate plate';
   aRecipe[2].RecipeCbsType := 'Carbody shell';
   aRecipe[3].RecipeCbsType := 'RGC';
   aRecipe[4..5].RecipeCbsType := '';
   aRecipe[7..23].RecipeCbsType := '';
   aRecipe[1].RecipeTrajNumber := 100;
   aRecipe[2].RecipeTrajNumber := 101;
   aRecipe[3].RecipeTrajNumber := 11;
   aRecipe[4..8].RecipeTrajNumber := 0;
   aRecipe[10..23].RecipeTrajNumber := 0;
   aRecipe[1..3].RecipeRawMaterial := 1;
   aRecipe[4..8].RecipeRawMaterial := 0;
   aRecipe[10..23].RecipeRawMaterial := 0;
   aRecipe[4].RecipeLayerType[1].RecipeLayerTypeName := '';
   aRecipe[5].RecipeLayerType[1].RecipeLayerTypeName := '';
   aRecipe[6].RecipeLayerType[1].RecipeLayerTypeName := '';
   aRecipe[7].RecipeLayerType[1].RecipeLayerTypeName := '';
   aRecipe[8].RecipeLayerType[1].RecipeLayerTypeName := '';
   aRecipe[9].RecipeLayerType[1].RecipeLayerTypeName := '';
   aRecipe[10].RecipeLayerType[1].RecipeLayerTypeName := '';
   aRecipe[11].RecipeLayerType[1].RecipeLayerTypeName := '';
   aRecipe[12].RecipeLayerType[1].RecipeLayerTypeName := '';
   aRecipe[13].RecipeLayerType[1].RecipeLayerTypeName := '';
   aRecipe[14].RecipeLayerType[1].RecipeLayerTypeName := '';
   aRecipe[15].RecipeLayerType[1].RecipeLayerTypeName := '';
   aRecipe[16].RecipeLayerType[1].RecipeLayerTypeName := '';
   aRecipe[17].RecipeLayerType[1].RecipeLayerTypeName := '';
   aRecipe[18].RecipeLayerType[1].RecipeLayerTypeName := '';
   aRecipe[19].RecipeLayerType[1].RecipeLayerTypeName := '';
   aRecipe[20].RecipeLayerType[1].RecipeLayerTypeName := '';
   aRecipe[21].RecipeLayerType[1].RecipeLayerTypeName := '';
   aRecipe[22].RecipeLayerType[1].RecipeLayerTypeName := '';
   aRecipe[23].RecipeLayerType[1].RecipeLayerTypeName := '';
   aRecipe[1].RecipeLayerType[1].JobTableLeft[0].SetForceZero := 0;
   aRecipe[1].RecipeLayerType[1].JobTableLeft[1..4].SetForceZero := 100;
   aRecipe[1].RecipeLayerType[2].JobTableLeft[0].SetForceZero := 0;
   aRecipe[1].RecipeLayerType[2].JobTableLeft[1].SetForceZero := 100;
   aRecipe[1].RecipeLayerType[2].JobTableLeft[2..3].SetForceZero := 90;
   aRecipe[2].RecipeLayerType[1].JobTableLeft[0].SetForceZero := 0;
   aRecipe[2].RecipeLayerType[1].JobTableLeft[1].SetForceZero := 50;
   aRecipe[2].RecipeLayerType[2].JobTableLeft[0].SetForceZero := 0;
   aRecipe[2].RecipeLayerType[2].JobTableLeft[1].SetForceZero := 100;
   aRecipe[2].RecipeLayerType[2].JobTableLeft[2..3].SetForceZero := 80;
   aRecipe[3].RecipeLayerType[1].JobTableLeft[0].SetForceZero := 0;
   aRecipe[3].RecipeLayerType[1].JobTableLeft[1..2].SetForceZero := 80;
   aRecipe[3].RecipeLayerType[2].JobTableLeft[0].SetForceZero := 0;
   aRecipe[3].RecipeLayerType[2].JobTableLeft[1].SetForceZero := 80;
   aRecipe[4].RecipeLayerType[1].JobTableLeft[0].SetForceZero := 0;
   aRecipe[4].RecipeLayerType[2].JobTableLeft[0].SetForceZero := 0;
   aRecipe[5].RecipeLayerType[1].JobTableLeft[0].SetForceZero := 0;
   aRecipe[5].RecipeLayerType[2].JobTableLeft[0].SetForceZero := 0;
   aRecipe[6].RecipeLayerType[1].JobTableLeft[0].SetForceZero := 0;
   aRecipe[6].RecipeLayerType[1].JobTableLeft[1].SetForceZero := 20;
   aRecipe[6].RecipeLayerType[2].JobTableLeft[0].SetForceZero := 0;
   aRecipe[6].RecipeLayerType[2].JobTableLeft[1].SetForceZero := 20;
   aRecipe[7].RecipeLayerType[1].JobTableLeft[0].SetForceZero := 0;
   aRecipe[7].RecipeLayerType[2].JobTableLeft[0].SetForceZero := 0;
   aRecipe[8].RecipeLayerType[1].JobTableLeft[0].SetForceZero := 0;
   aRecipe[8].RecipeLayerType[2].JobTableLeft[0].SetForceZero := 0;
   aRecipe[9].RecipeLayerType[1].JobTableLeft[0].SetForceZero := 0;
   aRecipe[9].RecipeLayerType[2].JobTableLeft[0].SetForceZero := 0;
   aRecipe[10].RecipeLayerType[1].JobTableLeft[0].SetForceZero := 0;
   aRecipe[10].RecipeLayerType[2].JobTableLeft[0].SetForceZero := 0;
   aRecipe[11].RecipeLayerType[1].JobTableLeft[0].SetForceZero := 0;
   aRecipe[11].RecipeLayerType[2].JobTableLeft[0].SetForceZero := 0;
   aRecipe[12].RecipeLayerType[1].JobTableLeft[0].SetForceZero := 0;
   aRecipe[12].RecipeLayerType[2].JobTableLeft[0].SetForceZero := 0;
   aRecipe[13].RecipeLayerType[1].JobTableLeft[0].SetForceZero := 0;
   aRecipe[13].RecipeLayerType[2].JobTableLeft[0].SetForceZero := 0;
   aRecipe[14].RecipeLayerType[1].JobTableLeft[0].SetForceZero := 0;
   aRecipe[14].RecipeLayerType[2].JobTableLeft[0].SetForceZero := 0;
   aRecipe[15].RecipeLayerType[1].JobTableLeft[0].SetForceZero := 0;
   aRecipe[15].RecipeLayerType[2].JobTableLeft[0].SetForceZero := 0;
   aRecipe[16].RecipeLayerType[1].JobTableLeft[0].SetForceZero := 0;
   aRecipe[16].RecipeLayerType[2].JobTableLeft[0].SetForceZero := 0;
   aRecipe[17].RecipeLayerType[1].JobTableLeft[0].SetForceZero := 0;
   aRecipe[17].RecipeLayerType[2].JobTableLeft[0].SetForceZero := 0;
   aRecipe[18].RecipeLayerType[1].JobTableLeft[0].SetForceZero := 0;
   aRecipe[18].RecipeLayerType[2].JobTableLeft[0].SetForceZero := 0;
   aRecipe[19].RecipeLayerType[1].JobTableLeft[0].SetForceZero := 0;
   aRecipe[19].RecipeLayerType[2].JobTableLeft[0].SetForceZero := 0;
   aRecipe[20].RecipeLayerType[1].JobTableLeft[0].SetForceZero := 0;
   aRecipe[20].RecipeLayerType[2].JobTableLeft[0].SetForceZero := 0;
   aRecipe[21].RecipeLayerType[1].JobTableLeft[0].SetForceZero := 0;
   aRecipe[21].RecipeLayerType[2].JobTableLeft[0].SetForceZero := 0;
   aRecipe[22].RecipeLayerType[1].JobTableLeft[0].SetForceZero := 0;
   aRecipe[22].RecipeLayerType[2].JobTableLeft[0].SetForceZero := 0;
   aRecipe[23].RecipeLayerType[1].JobTableLeft[0].SetForceZero := 0;
   aRecipe[23].RecipeLayerType[2].JobTableLeft[0].SetForceZero := 0;
   aRecipe[1].RecipeLayerType[1].JobTableLeft[0].SetForceTarget := 0;
   aRecipe[1].RecipeLayerType[1].JobTableLeft[1..4].SetForceTarget := 200;
   aRecipe[1].RecipeLayerType[2].JobTableLeft[0].SetForceTarget := 0;
   aRecipe[1].RecipeLayerType[2].JobTableLeft[1].SetForceTarget := 200;
   aRecipe[1].RecipeLayerType[2].JobTableLeft[2].SetForceTarget := 150;
   aRecipe[1].RecipeLayerType[2].JobTableLeft[3].SetForceTarget := 180;
   aRecipe[2].RecipeLayerType[1].JobTableLeft[0].SetForceTarget := 0;
   aRecipe[2].RecipeLayerType[1].JobTableLeft[1].SetForceTarget := 80;
   aRecipe[2].RecipeLayerType[2].JobTableLeft[0].SetForceTarget := 0;
   aRecipe[2].RecipeLayerType[2].JobTableLeft[1].SetForceTarget := 200;
   aRecipe[2].RecipeLayerType[2].JobTableLeft[3].SetForceTarget := 150;
   aRecipe[3].RecipeLayerType[1].JobTableLeft[0].SetForceTarget := 0;
   aRecipe[3].RecipeLayerType[1].JobTableLeft[1..2].SetForceTarget := 120;
   aRecipe[3].RecipeLayerType[2].JobTableLeft[0].SetForceTarget := 0;
   aRecipe[3].RecipeLayerType[2].JobTableLeft[1].SetForceTarget := 120;
   aRecipe[4].RecipeLayerType[1].JobTableLeft[0].SetForceTarget := 0;
   aRecipe[4].RecipeLayerType[2].JobTableLeft[0].SetForceTarget := 0;
   aRecipe[5].RecipeLayerType[1].JobTableLeft[0].SetForceTarget := 0;
   aRecipe[5].RecipeLayerType[2].JobTableLeft[0].SetForceTarget := 0;
   aRecipe[6].RecipeLayerType[1].JobTableLeft[0].SetForceTarget := 0;
   aRecipe[6].RecipeLayerType[1].JobTableLeft[1].SetForceTarget := 120;
   aRecipe[6].RecipeLayerType[2].JobTableLeft[0].SetForceTarget := 0;
   aRecipe[6].RecipeLayerType[2].JobTableLeft[1].SetForceTarget := 120;
   aRecipe[7].RecipeLayerType[1].JobTableLeft[0].SetForceTarget := 0;
   aRecipe[7].RecipeLayerType[2].JobTableLeft[0].SetForceTarget := 0;
   aRecipe[8].RecipeLayerType[1].JobTableLeft[0].SetForceTarget := 0;
   aRecipe[8].RecipeLayerType[2].JobTableLeft[0].SetForceTarget := 0;
   aRecipe[9].RecipeLayerType[1].JobTableLeft[0].SetForceTarget := 0;
   aRecipe[9].RecipeLayerType[2].JobTableLeft[0].SetForceTarget := 0;
   aRecipe[10].RecipeLayerType[1].JobTableLeft[0].SetForceTarget := 0;
   aRecipe[10].RecipeLayerType[2].JobTableLeft[0].SetForceTarget := 0;
   aRecipe[11].RecipeLayerType[1].JobTableLeft[0].SetForceTarget := 0;
   aRecipe[11].RecipeLayerType[2].JobTableLeft[0].SetForceTarget := 0;
   aRecipe[12].RecipeLayerType[1].JobTableLeft[0].SetForceTarget := 0;
   aRecipe[12].RecipeLayerType[2].JobTableLeft[0].SetForceTarget := 0;
   aRecipe[13].RecipeLayerType[1].JobTableLeft[0].SetForceTarget := 0;
   aRecipe[13].RecipeLayerType[2].JobTableLeft[0].SetForceTarget := 0;
   aRecipe[14].RecipeLayerType[1].JobTableLeft[0].SetForceTarget := 0;
   aRecipe[14].RecipeLayerType[2].JobTableLeft[0].SetForceTarget := 0;
   aRecipe[15].RecipeLayerType[1].JobTableLeft[0].SetForceTarget := 0;
   aRecipe[15].RecipeLayerType[2].JobTableLeft[0].SetForceTarget := 0;
   aRecipe[16].RecipeLayerType[1].JobTableLeft[0].SetForceTarget := 0;
   aRecipe[16].RecipeLayerType[2].JobTableLeft[0].SetForceTarget := 0;
   aRecipe[17].RecipeLayerType[1].JobTableLeft[0].SetForceTarget := 0;
   aRecipe[17].RecipeLayerType[2].JobTableLeft[0].SetForceTarget := 0;
   aRecipe[18].RecipeLayerType[1].JobTableLeft[0].SetForceTarget := 0;
   aRecipe[18].RecipeLayerType[2].JobTableLeft[0].SetForceTarget := 0;
   aRecipe[19].RecipeLayerType[1].JobTableLeft[0].SetForceTarget := 0;
   aRecipe[19].RecipeLayerType[2].JobTableLeft[0].SetForceTarget := 0;
   aRecipe[20].RecipeLayerType[1].JobTableLeft[0].SetForceTarget := 0;
   aRecipe[20].RecipeLayerType[2].JobTableLeft[0].SetForceTarget := 0;
   aRecipe[21].RecipeLayerType[1].JobTableLeft[0].SetForceTarget := 0;
   aRecipe[21].RecipeLayerType[2].JobTableLeft[0].SetForceTarget := 0;
   aRecipe[22].RecipeLayerType[1].JobTableLeft[0].SetForceTarget := 0;
   aRecipe[22].RecipeLayerType[2].JobTableLeft[0].SetForceTarget := 0;
   aRecipe[23].RecipeLayerType[1].JobTableLeft[0].SetForceTarget := 0;
   aRecipe[23].RecipeLayerType[2].JobTableLeft[0].SetForceTarget := 0;
   aRecipe[1].RecipeLayerType[1].JobTableLeft[0].SetTimeRamp := 0;
   aRecipe[1].RecipeLayerType[2].JobTableLeft[0].SetTimeRamp := 0;
   aRecipe[2].RecipeLayerType[1].JobTableLeft[0].SetTimeRamp := 0;
   aRecipe[2].RecipeLayerType[2].JobTableLeft[0].SetTimeRamp := 0;
   aRecipe[3].RecipeLayerType[1].JobTableLeft[0].SetTimeRamp := 0;
   aRecipe[3].RecipeLayerType[2].JobTableLeft[0].SetTimeRamp := 0;
   aRecipe[4].RecipeLayerType[1].JobTableLeft[0].SetTimeRamp := 0;
   aRecipe[4].RecipeLayerType[2].JobTableLeft[0].SetTimeRamp := 0;
   aRecipe[5].RecipeLayerType[1].JobTableLeft[0].SetTimeRamp := 0;
   aRecipe[5].RecipeLayerType[2].JobTableLeft[0].SetTimeRamp := 0;
   aRecipe[6].RecipeLayerType[1].JobTableLeft[0].SetTimeRamp := 0;
   aRecipe[6].RecipeLayerType[2].JobTableLeft[0].SetTimeRamp := 0;
   aRecipe[7].RecipeLayerType[1].JobTableLeft[0].SetTimeRamp := 0;
   aRecipe[7].RecipeLayerType[2].JobTableLeft[0].SetTimeRamp := 0;
   aRecipe[8].RecipeLayerType[1].JobTableLeft[0].SetTimeRamp := 0;
   aRecipe[8].RecipeLayerType[2].JobTableLeft[0].SetTimeRamp := 0;
   aRecipe[9].RecipeLayerType[1].JobTableLeft[0].SetTimeRamp := 0;
   aRecipe[9].RecipeLayerType[2].JobTableLeft[0].SetTimeRamp := 0;
   aRecipe[10].RecipeLayerType[1].JobTableLeft[0].SetTimeRamp := 0;
   aRecipe[10].RecipeLayerType[2].JobTableLeft[0].SetTimeRamp := 0;
   aRecipe[11].RecipeLayerType[1].JobTableLeft[0].SetTimeRamp := 0;
   aRecipe[11].RecipeLayerType[2].JobTableLeft[0].SetTimeRamp := 0;
   aRecipe[12].RecipeLayerType[1].JobTableLeft[0].SetTimeRamp := 0;
   aRecipe[12].RecipeLayerType[2].JobTableLeft[0].SetTimeRamp := 0;
   aRecipe[13].RecipeLayerType[1].JobTableLeft[0].SetTimeRamp := 0;
   aRecipe[13].RecipeLayerType[2].JobTableLeft[0].SetTimeRamp := 0;
   aRecipe[14].RecipeLayerType[1].JobTableLeft[0].SetTimeRamp := 0;
   aRecipe[14].RecipeLayerType[2].JobTableLeft[0].SetTimeRamp := 0;
   aRecipe[15].RecipeLayerType[1].JobTableLeft[0].SetTimeRamp := 0;
   aRecipe[15].RecipeLayerType[2].JobTableLeft[0].SetTimeRamp := 0;
   aRecipe[16].RecipeLayerType[1].JobTableLeft[0].SetTimeRamp := 0;
   aRecipe[16].RecipeLayerType[2].JobTableLeft[0].SetTimeRamp := 0;
   aRecipe[17].RecipeLayerType[1].JobTableLeft[0].SetTimeRamp := 0;
   aRecipe[17].RecipeLayerType[2].JobTableLeft[0].SetTimeRamp := 0;
   aRecipe[18].RecipeLayerType[1].JobTableLeft[0].SetTimeRamp := 0;
   aRecipe[18].RecipeLayerType[2].JobTableLeft[0].SetTimeRamp := 0;
   aRecipe[19].RecipeLayerType[1].JobTableLeft[0].SetTimeRamp := 0;
   aRecipe[19].RecipeLayerType[2].JobTableLeft[0].SetTimeRamp := 0;
   aRecipe[20].RecipeLayerType[1].JobTableLeft[0].SetTimeRamp := 0;
   aRecipe[20].RecipeLayerType[2].JobTableLeft[0].SetTimeRamp := 0;
   aRecipe[21].RecipeLayerType[1].JobTableLeft[0].SetTimeRamp := 0;
   aRecipe[21].RecipeLayerType[2].JobTableLeft[0].SetTimeRamp := 0;
   aRecipe[22].RecipeLayerType[1].JobTableLeft[0].SetTimeRamp := 0;
   aRecipe[22].RecipeLayerType[2].JobTableLeft[0].SetTimeRamp := 0;
   aRecipe[23].RecipeLayerType[1].JobTableLeft[0].SetTimeRamp := 0;
   aRecipe[23].RecipeLayerType[2].JobTableLeft[0].SetTimeRamp := 0;
   aRecipe[1].RecipeLayerType[1].JobTableLeft[0].SetSpeed := 0;
   aRecipe[1].RecipeLayerType[1].JobTableLeft[3..4].SetSpeed := 5000;
   aRecipe[1].RecipeLayerType[2].JobTableLeft[0].SetSpeed := 0;
   aRecipe[2].RecipeLayerType[1].JobTableLeft[0].SetSpeed := 0;
   aRecipe[2].RecipeLayerType[2].JobTableLeft[0].SetSpeed := 0;
   aRecipe[3].RecipeLayerType[1].JobTableLeft[0].SetSpeed := 0;
   aRecipe[3].RecipeLayerType[2].JobTableLeft[0].SetSpeed := 0;
   aRecipe[4].RecipeLayerType[1].JobTableLeft[0].SetSpeed := 0;
   aRecipe[4].RecipeLayerType[2].JobTableLeft[0].SetSpeed := 0;
   aRecipe[5].RecipeLayerType[1].JobTableLeft[0].SetSpeed := 0;
   aRecipe[5].RecipeLayerType[2].JobTableLeft[0].SetSpeed := 0;
   aRecipe[6].RecipeLayerType[1].JobTableLeft[0].SetSpeed := 0;
   aRecipe[6].RecipeLayerType[2].JobTableLeft[0].SetSpeed := 0;
   aRecipe[7].RecipeLayerType[1].JobTableLeft[0].SetSpeed := 0;
   aRecipe[7].RecipeLayerType[2].JobTableLeft[0].SetSpeed := 0;
   aRecipe[8].RecipeLayerType[1].JobTableLeft[0].SetSpeed := 0;
   aRecipe[8].RecipeLayerType[2].JobTableLeft[0].SetSpeed := 0;
   aRecipe[9].RecipeLayerType[1].JobTableLeft[0].SetSpeed := 0;
   aRecipe[9].RecipeLayerType[2].JobTableLeft[0].SetSpeed := 0;
   aRecipe[10].RecipeLayerType[1].JobTableLeft[0].SetSpeed := 0;
   aRecipe[10].RecipeLayerType[2].JobTableLeft[0].SetSpeed := 0;
   aRecipe[11].RecipeLayerType[1].JobTableLeft[0].SetSpeed := 0;
   aRecipe[11].RecipeLayerType[2].JobTableLeft[0].SetSpeed := 0;
   aRecipe[12].RecipeLayerType[1].JobTableLeft[0].SetSpeed := 0;
   aRecipe[12].RecipeLayerType[2].JobTableLeft[0].SetSpeed := 0;
   aRecipe[13].RecipeLayerType[1].JobTableLeft[0].SetSpeed := 0;
   aRecipe[13].RecipeLayerType[2].JobTableLeft[0].SetSpeed := 0;
   aRecipe[14].RecipeLayerType[1].JobTableLeft[0].SetSpeed := 0;
   aRecipe[14].RecipeLayerType[2].JobTableLeft[0].SetSpeed := 0;
   aRecipe[15].RecipeLayerType[1].JobTableLeft[0].SetSpeed := 0;
   aRecipe[15].RecipeLayerType[2].JobTableLeft[0].SetSpeed := 0;
   aRecipe[16].RecipeLayerType[1].JobTableLeft[0].SetSpeed := 0;
   aRecipe[16].RecipeLayerType[2].JobTableLeft[0].SetSpeed := 0;
   aRecipe[17].RecipeLayerType[1].JobTableLeft[0].SetSpeed := 0;
   aRecipe[17].RecipeLayerType[2].JobTableLeft[0].SetSpeed := 0;
   aRecipe[18].RecipeLayerType[1].JobTableLeft[0].SetSpeed := 0;
   aRecipe[18].RecipeLayerType[2].JobTableLeft[0].SetSpeed := 0;
   aRecipe[19].RecipeLayerType[1].JobTableLeft[0].SetSpeed := 0;
   aRecipe[19].RecipeLayerType[2].JobTableLeft[0].SetSpeed := 0;
   aRecipe[20].RecipeLayerType[1].JobTableLeft[0].SetSpeed := 0;
   aRecipe[20].RecipeLayerType[2].JobTableLeft[0].SetSpeed := 0;
   aRecipe[21].RecipeLayerType[1].JobTableLeft[0].SetSpeed := 0;
   aRecipe[21].RecipeLayerType[2].JobTableLeft[0].SetSpeed := 0;
   aRecipe[22].RecipeLayerType[1].JobTableLeft[0].SetSpeed := 0;
   aRecipe[22].RecipeLayerType[2].JobTableLeft[0].SetSpeed := 0;
   aRecipe[23].RecipeLayerType[1].JobTableLeft[0].SetSpeed := 0;
   aRecipe[23].RecipeLayerType[2].JobTableLeft[0].SetSpeed := 0;
   aRecipe[1].RecipeLayerType[1].JobTableLeft[0].SetRobotSpeed := 0;
   aRecipe[1].RecipeLayerType[1].JobTableLeft[1].SetRobotSpeed := 300;
   aRecipe[1].RecipeLayerType[1].JobTableLeft[2].SetRobotSpeed := 500;
   aRecipe[1].RecipeLayerType[1].JobTableLeft[3..4].SetRobotSpeed := 300;
   aRecipe[1].RecipeLayerType[2].JobTableLeft[0].SetRobotSpeed := 0;
   aRecipe[1].RecipeLayerType[2].JobTableLeft[1..3].SetRobotSpeed := 300;
   aRecipe[2].RecipeLayerType[1].JobTableLeft[0].SetRobotSpeed := 0;
   aRecipe[2].RecipeLayerType[1].JobTableLeft[1].SetRobotSpeed := 300;
   aRecipe[2].RecipeLayerType[2].JobTableLeft[0].SetRobotSpeed := 0;
   aRecipe[2].RecipeLayerType[2].JobTableLeft[1..2].SetRobotSpeed := 300;
   aRecipe[2].RecipeLayerType[2].JobTableLeft[3].SetRobotSpeed := 250;
   aRecipe[3].RecipeLayerType[1].JobTableLeft[0].SetRobotSpeed := 0;
   aRecipe[3].RecipeLayerType[1].JobTableLeft[1].SetRobotSpeed := 200;
   aRecipe[3].RecipeLayerType[1].JobTableLeft[2].SetRobotSpeed := 300;
   aRecipe[3].RecipeLayerType[2].JobTableLeft[0].SetRobotSpeed := 0;
   aRecipe[3].RecipeLayerType[2].JobTableLeft[1].SetRobotSpeed := 300;
   aRecipe[4].RecipeLayerType[1].JobTableLeft[0].SetRobotSpeed := 0;
   aRecipe[4].RecipeLayerType[2].JobTableLeft[0].SetRobotSpeed := 0;
   aRecipe[5].RecipeLayerType[1].JobTableLeft[0].SetRobotSpeed := 0;
   aRecipe[5].RecipeLayerType[2].JobTableLeft[0].SetRobotSpeed := 0;
   aRecipe[6].RecipeLayerType[1].JobTableLeft[0].SetRobotSpeed := 0;
   aRecipe[6].RecipeLayerType[2].JobTableLeft[0].SetRobotSpeed := 0;
   aRecipe[7].RecipeLayerType[1].JobTableLeft[0].SetRobotSpeed := 0;
   aRecipe[7].RecipeLayerType[2].JobTableLeft[0].SetRobotSpeed := 0;
   aRecipe[8].RecipeLayerType[1].JobTableLeft[0].SetRobotSpeed := 0;
   aRecipe[8].RecipeLayerType[2].JobTableLeft[0].SetRobotSpeed := 0;
   aRecipe[9].RecipeLayerType[1].JobTableLeft[0].SetRobotSpeed := 0;
   aRecipe[9].RecipeLayerType[2].JobTableLeft[0].SetRobotSpeed := 0;
   aRecipe[10].RecipeLayerType[1].JobTableLeft[0].SetRobotSpeed := 0;
   aRecipe[10].RecipeLayerType[2].JobTableLeft[0].SetRobotSpeed := 0;
   aRecipe[11].RecipeLayerType[1].JobTableLeft[0].SetRobotSpeed := 0;
   aRecipe[11].RecipeLayerType[2].JobTableLeft[0].SetRobotSpeed := 0;
   aRecipe[12].RecipeLayerType[1].JobTableLeft[0].SetRobotSpeed := 0;
   aRecipe[12].RecipeLayerType[2].JobTableLeft[0].SetRobotSpeed := 0;
   aRecipe[13].RecipeLayerType[1].JobTableLeft[0].SetRobotSpeed := 0;
   aRecipe[13].RecipeLayerType[2].JobTableLeft[0].SetRobotSpeed := 0;
   aRecipe[14].RecipeLayerType[1].JobTableLeft[0].SetRobotSpeed := 0;
   aRecipe[14].RecipeLayerType[2].JobTableLeft[0].SetRobotSpeed := 0;
   aRecipe[15].RecipeLayerType[1].JobTableLeft[0].SetRobotSpeed := 0;
   aRecipe[15].RecipeLayerType[2].JobTableLeft[0].SetRobotSpeed := 0;
   aRecipe[16].RecipeLayerType[1].JobTableLeft[0].SetRobotSpeed := 0;
   aRecipe[16].RecipeLayerType[2].JobTableLeft[0].SetRobotSpeed := 0;
   aRecipe[17].RecipeLayerType[1].JobTableLeft[0].SetRobotSpeed := 0;
   aRecipe[17].RecipeLayerType[2].JobTableLeft[0].SetRobotSpeed := 0;
   aRecipe[18].RecipeLayerType[1].JobTableLeft[0].SetRobotSpeed := 0;
   aRecipe[18].RecipeLayerType[2].JobTableLeft[0].SetRobotSpeed := 0;
   aRecipe[19].RecipeLayerType[1].JobTableLeft[0].SetRobotSpeed := 0;
   aRecipe[19].RecipeLayerType[2].JobTableLeft[0].SetRobotSpeed := 0;
   aRecipe[20].RecipeLayerType[1].JobTableLeft[0].SetRobotSpeed := 0;
   aRecipe[20].RecipeLayerType[2].JobTableLeft[0].SetRobotSpeed := 0;
   aRecipe[21].RecipeLayerType[1].JobTableLeft[0].SetRobotSpeed := 0;
   aRecipe[21].RecipeLayerType[2].JobTableLeft[0].SetRobotSpeed := 0;
   aRecipe[22].RecipeLayerType[1].JobTableLeft[0].SetRobotSpeed := 0;
   aRecipe[22].RecipeLayerType[2].JobTableLeft[0].SetRobotSpeed := 0;
   aRecipe[23].RecipeLayerType[1].JobTableLeft[0].SetRobotSpeed := 0;
   aRecipe[23].RecipeLayerType[2].JobTableLeft[0].SetRobotSpeed := 0;
   aRecipe[1].RecipeLayerType[1].JobTableLeft[0].WornPaperDistance := 0;
   aRecipe[1].RecipeLayerType[1].JobTableLeft[1..4].WornPaperDistance := 900;
   aRecipe[1].RecipeLayerType[2].JobTableLeft[0].WornPaperDistance := 0;
   aRecipe[1].RecipeLayerType[2].JobTableLeft[1..3].WornPaperDistance := 900;
   aRecipe[2].RecipeLayerType[1].JobTableLeft[0].WornPaperDistance := 0;
   aRecipe[2].RecipeLayerType[1].JobTableLeft[1].WornPaperDistance := 8;
   aRecipe[2].RecipeLayerType[1].JobTableLeft[2..3].WornPaperDistance := 999;
   aRecipe[2].RecipeLayerType[2].JobTableLeft[0].WornPaperDistance := 0;
   aRecipe[2].RecipeLayerType[2].JobTableLeft[1..2].WornPaperDistance := 30;
   aRecipe[2].RecipeLayerType[2].JobTableLeft[3].WornPaperDistance := 999;
   aRecipe[3].RecipeLayerType[1].JobTableLeft[0].WornPaperDistance := 0;
   aRecipe[3].RecipeLayerType[1].JobTableLeft[1..2].WornPaperDistance := 30;
   aRecipe[3].RecipeLayerType[2].JobTableLeft[0].WornPaperDistance := 0;
   aRecipe[3].RecipeLayerType[2].JobTableLeft[1].WornPaperDistance := 30;
   aRecipe[4].RecipeLayerType[1].JobTableLeft[0].WornPaperDistance := 0;
   aRecipe[4].RecipeLayerType[2].JobTableLeft[0].WornPaperDistance := 0;
   aRecipe[5].RecipeLayerType[1].JobTableLeft[0].WornPaperDistance := 0;
   aRecipe[5].RecipeLayerType[2].JobTableLeft[0].WornPaperDistance := 0;
   aRecipe[6].RecipeLayerType[1].JobTableLeft[0].WornPaperDistance := 0;
   aRecipe[6].RecipeLayerType[2].JobTableLeft[0].WornPaperDistance := 0;
   aRecipe[7].RecipeLayerType[1].JobTableLeft[0].WornPaperDistance := 0;
   aRecipe[7].RecipeLayerType[2].JobTableLeft[0].WornPaperDistance := 0;
   aRecipe[8].RecipeLayerType[1].JobTableLeft[0].WornPaperDistance := 0;
   aRecipe[8].RecipeLayerType[2].JobTableLeft[0].WornPaperDistance := 0;
   aRecipe[9].RecipeLayerType[1].JobTableLeft[0].WornPaperDistance := 0;
   aRecipe[9].RecipeLayerType[2].JobTableLeft[0].WornPaperDistance := 0;
   aRecipe[10].RecipeLayerType[1].JobTableLeft[0].WornPaperDistance := 0;
   aRecipe[10].RecipeLayerType[2].JobTableLeft[0].WornPaperDistance := 0;
   aRecipe[11].RecipeLayerType[1].JobTableLeft[0].WornPaperDistance := 0;
   aRecipe[11].RecipeLayerType[2].JobTableLeft[0].WornPaperDistance := 0;
   aRecipe[12].RecipeLayerType[1].JobTableLeft[0].WornPaperDistance := 0;
   aRecipe[12].RecipeLayerType[2].JobTableLeft[0].WornPaperDistance := 0;
   aRecipe[13].RecipeLayerType[1].JobTableLeft[0].WornPaperDistance := 0;
   aRecipe[13].RecipeLayerType[2].JobTableLeft[0].WornPaperDistance := 0;
   aRecipe[14].RecipeLayerType[1].JobTableLeft[0].WornPaperDistance := 0;
   aRecipe[14].RecipeLayerType[2].JobTableLeft[0].WornPaperDistance := 0;
   aRecipe[15].RecipeLayerType[1].JobTableLeft[0].WornPaperDistance := 0;
   aRecipe[15].RecipeLayerType[2].JobTableLeft[0].WornPaperDistance := 0;
   aRecipe[16].RecipeLayerType[1].JobTableLeft[0].WornPaperDistance := 0;
   aRecipe[16].RecipeLayerType[2].JobTableLeft[0].WornPaperDistance := 0;
   aRecipe[17].RecipeLayerType[1].JobTableLeft[0].WornPaperDistance := 0;
   aRecipe[17].RecipeLayerType[2].JobTableLeft[0].WornPaperDistance := 0;
   aRecipe[18].RecipeLayerType[1].JobTableLeft[0].WornPaperDistance := 0;
   aRecipe[18].RecipeLayerType[2].JobTableLeft[0].WornPaperDistance := 0;
   aRecipe[19].RecipeLayerType[1].JobTableLeft[0].WornPaperDistance := 0;
   aRecipe[19].RecipeLayerType[2].JobTableLeft[0].WornPaperDistance := 0;
   aRecipe[20].RecipeLayerType[1].JobTableLeft[0].WornPaperDistance := 0;
   aRecipe[20].RecipeLayerType[2].JobTableLeft[0].WornPaperDistance := 0;
   aRecipe[21].RecipeLayerType[1].JobTableLeft[0].WornPaperDistance := 0;
   aRecipe[21].RecipeLayerType[2].JobTableLeft[0].WornPaperDistance := 0;
   aRecipe[22].RecipeLayerType[1].JobTableLeft[0].WornPaperDistance := 0;
   aRecipe[22].RecipeLayerType[2].JobTableLeft[0].WornPaperDistance := 0;
   aRecipe[23].RecipeLayerType[1].JobTableLeft[0].WornPaperDistance := 0;
   aRecipe[23].RecipeLayerType[2].JobTableLeft[0].WornPaperDistance := 0;
   aRecipe[1].RecipeLayerType[1].JobTableLeft[0].Gimball := 0;
   aRecipe[1].RecipeLayerType[2].JobTableLeft[0].Gimball := 0;
   aRecipe[2].RecipeLayerType[1].JobTableLeft[0].Gimball := 0;
   aRecipe[2].RecipeLayerType[2].JobTableLeft[0].Gimball := 0;
   aRecipe[3].RecipeLayerType[1].JobTableLeft[0].Gimball := 0;
   aRecipe[3].RecipeLayerType[2].JobTableLeft[0].Gimball := 0;
   aRecipe[3].RecipeLayerType[2].JobTableLeft[1].Gimball := 1;
   aRecipe[4].RecipeLayerType[1].JobTableLeft[0].Gimball := 0;
   aRecipe[4].RecipeLayerType[2].JobTableLeft[0].Gimball := 0;
   aRecipe[5].RecipeLayerType[1].JobTableLeft[0].Gimball := 0;
   aRecipe[5].RecipeLayerType[2].JobTableLeft[0].Gimball := 0;
   aRecipe[6].RecipeLayerType[1].JobTableLeft[0].Gimball := 0;
   aRecipe[6].RecipeLayerType[2].JobTableLeft[0].Gimball := 0;
   aRecipe[7].RecipeLayerType[1].JobTableLeft[0].Gimball := 0;
   aRecipe[7].RecipeLayerType[2].JobTableLeft[0].Gimball := 0;
   aRecipe[8].RecipeLayerType[1].JobTableLeft[0].Gimball := 0;
   aRecipe[8].RecipeLayerType[2].JobTableLeft[0].Gimball := 0;
   aRecipe[9].RecipeLayerType[1].JobTableLeft[0].Gimball := 0;
   aRecipe[9].RecipeLayerType[2].JobTableLeft[0].Gimball := 0;
   aRecipe[10].RecipeLayerType[1].JobTableLeft[0].Gimball := 0;
   aRecipe[10].RecipeLayerType[2].JobTableLeft[0].Gimball := 0;
   aRecipe[11].RecipeLayerType[1].JobTableLeft[0].Gimball := 0;
   aRecipe[11].RecipeLayerType[2].JobTableLeft[0].Gimball := 0;
   aRecipe[12].RecipeLayerType[1].JobTableLeft[0].Gimball := 0;
   aRecipe[12].RecipeLayerType[2].JobTableLeft[0].Gimball := 0;
   aRecipe[13].RecipeLayerType[1].JobTableLeft[0].Gimball := 0;
   aRecipe[13].RecipeLayerType[2].JobTableLeft[0].Gimball := 0;
   aRecipe[14].RecipeLayerType[1].JobTableLeft[0].Gimball := 0;
   aRecipe[14].RecipeLayerType[2].JobTableLeft[0].Gimball := 0;
   aRecipe[15].RecipeLayerType[1].JobTableLeft[0].Gimball := 0;
   aRecipe[15].RecipeLayerType[2].JobTableLeft[0].Gimball := 0;
   aRecipe[16].RecipeLayerType[1].JobTableLeft[0].Gimball := 0;
   aRecipe[16].RecipeLayerType[2].JobTableLeft[0].Gimball := 0;
   aRecipe[17].RecipeLayerType[1].JobTableLeft[0].Gimball := 0;
   aRecipe[17].RecipeLayerType[1].JobTableLeft[1].Gimball := 1;
   aRecipe[17].RecipeLayerType[2].JobTableLeft[0].Gimball := 0;
   aRecipe[18].RecipeLayerType[1].JobTableLeft[0].Gimball := 0;
   aRecipe[18].RecipeLayerType[2].JobTableLeft[0].Gimball := 0;
   aRecipe[19].RecipeLayerType[1].JobTableLeft[0].Gimball := 0;
   aRecipe[19].RecipeLayerType[2].JobTableLeft[0].Gimball := 0;
   aRecipe[20].RecipeLayerType[1].JobTableLeft[0].Gimball := 0;
   aRecipe[20].RecipeLayerType[2].JobTableLeft[0].Gimball := 0;
   aRecipe[21].RecipeLayerType[1].JobTableLeft[0].Gimball := 0;
   aRecipe[21].RecipeLayerType[2].JobTableLeft[0].Gimball := 0;
   aRecipe[22].RecipeLayerType[1].JobTableLeft[0].Gimball := 0;
   aRecipe[22].RecipeLayerType[2].JobTableLeft[0].Gimball := 0;
   aRecipe[23].RecipeLayerType[1].JobTableLeft[0].Gimball := 0;
   aRecipe[23].RecipeLayerType[2].JobTableLeft[0].Gimball := 0;
   aRecipe[1].RecipeLayerType[1].JobTableLeft[1..4].UnlockEccentric1 := TRUE;
   aRecipe[1].RecipeLayerType[2].JobTableLeft[3].UnlockEccentric1 := TRUE;
   aRecipe[1].RecipeLayerType[1].JobTableLeft[1..4].UnlockEccentric2 := TRUE;
   aRecipe[1].RecipeLayerType[2].JobTableLeft[3].UnlockEccentric2 := TRUE;
   aRecipe[1].RecipeLayerType[1].JobTableLeft[1..4].UnlockEccentric3 := TRUE;
   aRecipe[1].RecipeLayerType[2].JobTableLeft[3].UnlockEccentric3 := TRUE;
   aRecipe[1].RecipeLayerType[1].JobTableRight[0].SetForceZero := 0;
   aRecipe[1].RecipeLayerType[1].JobTableRight[1].SetForceZero := 21;
   aRecipe[1].RecipeLayerType[1].JobTableRight[2].SetForceZero := 22;
   aRecipe[1].RecipeLayerType[2].JobTableRight[0].SetForceZero := 0;
   aRecipe[2].RecipeLayerType[1].JobTableRight[0].SetForceZero := 0;
   aRecipe[2].RecipeLayerType[1].JobTableRight[1].SetForceZero := 50;
   aRecipe[2].RecipeLayerType[1].JobTableRight[2].SetForceZero := 80;
   aRecipe[2].RecipeLayerType[1].JobTableRight[3].SetForceZero := 50;
   aRecipe[2].RecipeLayerType[2].JobTableRight[0].SetForceZero := 0;
   aRecipe[2].RecipeLayerType[2].JobTableRight[1].SetForceZero := 100;
   aRecipe[2].RecipeLayerType[2].JobTableRight[2].SetForceZero := 80;
   aRecipe[3].RecipeLayerType[1].JobTableRight[0].SetForceZero := 0;
   aRecipe[3].RecipeLayerType[1].JobTableRight[1..2].SetForceZero := 80;
   aRecipe[3].RecipeLayerType[2].JobTableRight[0].SetForceZero := 0;
   aRecipe[3].RecipeLayerType[2].JobTableRight[1].SetForceZero := 80;
   aRecipe[4].RecipeLayerType[1].JobTableRight[0].SetForceZero := 0;
   aRecipe[4].RecipeLayerType[2].JobTableRight[0].SetForceZero := 0;
   aRecipe[5].RecipeLayerType[1].JobTableRight[0].SetForceZero := 0;
   aRecipe[5].RecipeLayerType[2].JobTableRight[0].SetForceZero := 0;
   aRecipe[6].RecipeLayerType[1].JobTableRight[0].SetForceZero := 0;
   aRecipe[6].RecipeLayerType[1].JobTableRight[1].SetForceZero := 20;
   aRecipe[6].RecipeLayerType[2].JobTableRight[0].SetForceZero := 0;
   aRecipe[6].RecipeLayerType[2].JobTableRight[1].SetForceZero := 20;
   aRecipe[7].RecipeLayerType[1].JobTableRight[0].SetForceZero := 0;
   aRecipe[7].RecipeLayerType[2].JobTableRight[0].SetForceZero := 0;
   aRecipe[8].RecipeLayerType[1].JobTableRight[0].SetForceZero := 0;
   aRecipe[8].RecipeLayerType[2].JobTableRight[0].SetForceZero := 0;
   aRecipe[9].RecipeLayerType[1].JobTableRight[0].SetForceZero := 0;
   aRecipe[9].RecipeLayerType[2].JobTableRight[0].SetForceZero := 0;
   aRecipe[10].RecipeLayerType[1].JobTableRight[0].SetForceZero := 0;
   aRecipe[10].RecipeLayerType[2].JobTableRight[0].SetForceZero := 0;
   aRecipe[11].RecipeLayerType[1].JobTableRight[0].SetForceZero := 0;
   aRecipe[11].RecipeLayerType[2].JobTableRight[0].SetForceZero := 0;
   aRecipe[12].RecipeLayerType[1].JobTableRight[0].SetForceZero := 0;
   aRecipe[12].RecipeLayerType[2].JobTableRight[0].SetForceZero := 0;
   aRecipe[13].RecipeLayerType[1].JobTableRight[0].SetForceZero := 0;
   aRecipe[13].RecipeLayerType[2].JobTableRight[0].SetForceZero := 0;
   aRecipe[14].RecipeLayerType[1].JobTableRight[0].SetForceZero := 0;
   aRecipe[14].RecipeLayerType[2].JobTableRight[0].SetForceZero := 0;
   aRecipe[15].RecipeLayerType[1].JobTableRight[0].SetForceZero := 0;
   aRecipe[15].RecipeLayerType[2].JobTableRight[0].SetForceZero := 0;
   aRecipe[16].RecipeLayerType[1].JobTableRight[0].SetForceZero := 0;
   aRecipe[16].RecipeLayerType[2].JobTableRight[0].SetForceZero := 0;
   aRecipe[17].RecipeLayerType[1].JobTableRight[0].SetForceZero := 0;
   aRecipe[17].RecipeLayerType[1].JobTableRight[1].SetForceZero := 20;
   aRecipe[17].RecipeLayerType[2].JobTableRight[0].SetForceZero := 0;
   aRecipe[18].RecipeLayerType[1].JobTableRight[0].SetForceZero := 0;
   aRecipe[18].RecipeLayerType[2].JobTableRight[0].SetForceZero := 0;
   aRecipe[19].RecipeLayerType[1].JobTableRight[0].SetForceZero := 0;
   aRecipe[19].RecipeLayerType[2].JobTableRight[0].SetForceZero := 0;
   aRecipe[20].RecipeLayerType[1].JobTableRight[0].SetForceZero := 0;
   aRecipe[20].RecipeLayerType[2].JobTableRight[0].SetForceZero := 0;
   aRecipe[21].RecipeLayerType[1].JobTableRight[0].SetForceZero := 0;
   aRecipe[21].RecipeLayerType[2].JobTableRight[0].SetForceZero := 0;
   aRecipe[22].RecipeLayerType[1].JobTableRight[0].SetForceZero := 0;
   aRecipe[22].RecipeLayerType[2].JobTableRight[0].SetForceZero := 0;
   aRecipe[23].RecipeLayerType[1].JobTableRight[0].SetForceZero := 0;
   aRecipe[23].RecipeLayerType[2].JobTableRight[0].SetForceZero := 0;
   aRecipe[1].RecipeLayerType[1].JobTableRight[0].SetForceTarget := 0;
   aRecipe[1].RecipeLayerType[2].JobTableRight[0].SetForceTarget := 0;
   aRecipe[2].RecipeLayerType[1].JobTableRight[0].SetForceTarget := 0;
   aRecipe[2].RecipeLayerType[1].JobTableRight[1].SetForceTarget := 80;
   aRecipe[2].RecipeLayerType[1].JobTableRight[3].SetForceTarget := 100;
   aRecipe[2].RecipeLayerType[2].JobTableRight[0].SetForceTarget := 0;
   aRecipe[2].RecipeLayerType[2].JobTableRight[1].SetForceTarget := 200;
   aRecipe[3].RecipeLayerType[1].JobTableRight[0].SetForceTarget := 0;
   aRecipe[3].RecipeLayerType[1].JobTableRight[1].SetForceTarget := 120;
   aRecipe[3].RecipeLayerType[2].JobTableRight[0].SetForceTarget := 0;
   aRecipe[3].RecipeLayerType[2].JobTableRight[1].SetForceTarget := 120;
   aRecipe[4].RecipeLayerType[1].JobTableRight[0].SetForceTarget := 0;
   aRecipe[4].RecipeLayerType[2].JobTableRight[0].SetForceTarget := 0;
   aRecipe[5].RecipeLayerType[1].JobTableRight[0].SetForceTarget := 0;
   aRecipe[5].RecipeLayerType[2].JobTableRight[0].SetForceTarget := 0;
   aRecipe[6].RecipeLayerType[1].JobTableRight[0].SetForceTarget := 0;
   aRecipe[6].RecipeLayerType[1].JobTableRight[1].SetForceTarget := 120;
   aRecipe[6].RecipeLayerType[2].JobTableRight[0].SetForceTarget := 0;
   aRecipe[6].RecipeLayerType[2].JobTableRight[1].SetForceTarget := 120;
   aRecipe[7].RecipeLayerType[1].JobTableRight[0].SetForceTarget := 0;
   aRecipe[7].RecipeLayerType[2].JobTableRight[0].SetForceTarget := 0;
   aRecipe[8].RecipeLayerType[1].JobTableRight[0].SetForceTarget := 0;
   aRecipe[8].RecipeLayerType[2].JobTableRight[0].SetForceTarget := 0;
   aRecipe[9].RecipeLayerType[1].JobTableRight[0].SetForceTarget := 0;
   aRecipe[9].RecipeLayerType[2].JobTableRight[0].SetForceTarget := 0;
   aRecipe[10].RecipeLayerType[1].JobTableRight[0].SetForceTarget := 0;
   aRecipe[10].RecipeLayerType[2].JobTableRight[0].SetForceTarget := 0;
   aRecipe[11].RecipeLayerType[1].JobTableRight[0].SetForceTarget := 0;
   aRecipe[11].RecipeLayerType[2].JobTableRight[0].SetForceTarget := 0;
   aRecipe[12].RecipeLayerType[1].JobTableRight[0].SetForceTarget := 0;
   aRecipe[12].RecipeLayerType[2].JobTableRight[0].SetForceTarget := 0;
   aRecipe[13].RecipeLayerType[1].JobTableRight[0].SetForceTarget := 0;
   aRecipe[13].RecipeLayerType[2].JobTableRight[0].SetForceTarget := 0;
   aRecipe[14].RecipeLayerType[1].JobTableRight[0].SetForceTarget := 0;
   aRecipe[14].RecipeLayerType[2].JobTableRight[0].SetForceTarget := 0;
   aRecipe[15].RecipeLayerType[1].JobTableRight[0].SetForceTarget := 0;
   aRecipe[15].RecipeLayerType[2].JobTableRight[0].SetForceTarget := 0;
   aRecipe[16].RecipeLayerType[1].JobTableRight[0].SetForceTarget := 0;
   aRecipe[16].RecipeLayerType[2].JobTableRight[0].SetForceTarget := 0;
   aRecipe[17].RecipeLayerType[1].JobTableRight[0].SetForceTarget := 0;
   aRecipe[17].RecipeLayerType[1].JobTableRight[1].SetForceTarget := 120;
   aRecipe[17].RecipeLayerType[2].JobTableRight[0].SetForceTarget := 0;
   aRecipe[18].RecipeLayerType[1].JobTableRight[0].SetForceTarget := 0;
   aRecipe[18].RecipeLayerType[2].JobTableRight[0].SetForceTarget := 0;
   aRecipe[19].RecipeLayerType[1].JobTableRight[0].SetForceTarget := 0;
   aRecipe[19].RecipeLayerType[2].JobTableRight[0].SetForceTarget := 0;
   aRecipe[20].RecipeLayerType[1].JobTableRight[0].SetForceTarget := 0;
   aRecipe[20].RecipeLayerType[2].JobTableRight[0].SetForceTarget := 0;
   aRecipe[21].RecipeLayerType[1].JobTableRight[0].SetForceTarget := 0;
   aRecipe[21].RecipeLayerType[2].JobTableRight[0].SetForceTarget := 0;
   aRecipe[22].RecipeLayerType[1].JobTableRight[0].SetForceTarget := 0;
   aRecipe[22].RecipeLayerType[2].JobTableRight[0].SetForceTarget := 0;
   aRecipe[23].RecipeLayerType[1].JobTableRight[0].SetForceTarget := 0;
   aRecipe[23].RecipeLayerType[2].JobTableRight[0].SetForceTarget := 0;
   aRecipe[1].RecipeLayerType[1].JobTableRight[0].SetTimeRamp := 0;
   aRecipe[1].RecipeLayerType[2].JobTableRight[0].SetTimeRamp := 0;
   aRecipe[2].RecipeLayerType[1].JobTableRight[0].SetTimeRamp := 0;
   aRecipe[2].RecipeLayerType[2].JobTableRight[0].SetTimeRamp := 0;
   aRecipe[3].RecipeLayerType[1].JobTableRight[0].SetTimeRamp := 0;
   aRecipe[3].RecipeLayerType[2].JobTableRight[0].SetTimeRamp := 0;
   aRecipe[4].RecipeLayerType[1].JobTableRight[0].SetTimeRamp := 0;
   aRecipe[4].RecipeLayerType[2].JobTableRight[0].SetTimeRamp := 0;
   aRecipe[5].RecipeLayerType[1].JobTableRight[0].SetTimeRamp := 0;
   aRecipe[5].RecipeLayerType[2].JobTableRight[0].SetTimeRamp := 0;
   aRecipe[6].RecipeLayerType[1].JobTableRight[0].SetTimeRamp := 0;
   aRecipe[6].RecipeLayerType[2].JobTableRight[0].SetTimeRamp := 0;
   aRecipe[7].RecipeLayerType[1].JobTableRight[0].SetTimeRamp := 0;
   aRecipe[7].RecipeLayerType[2].JobTableRight[0].SetTimeRamp := 0;
   aRecipe[8].RecipeLayerType[1].JobTableRight[0].SetTimeRamp := 0;
   aRecipe[8].RecipeLayerType[2].JobTableRight[0].SetTimeRamp := 0;
   aRecipe[9].RecipeLayerType[1].JobTableRight[0].SetTimeRamp := 0;
   aRecipe[9].RecipeLayerType[2].JobTableRight[0].SetTimeRamp := 0;
   aRecipe[10].RecipeLayerType[1].JobTableRight[0].SetTimeRamp := 0;
   aRecipe[10].RecipeLayerType[2].JobTableRight[0].SetTimeRamp := 0;
   aRecipe[11].RecipeLayerType[1].JobTableRight[0].SetTimeRamp := 0;
   aRecipe[11].RecipeLayerType[2].JobTableRight[0].SetTimeRamp := 0;
   aRecipe[12].RecipeLayerType[1].JobTableRight[0].SetTimeRamp := 0;
   aRecipe[12].RecipeLayerType[2].JobTableRight[0].SetTimeRamp := 0;
   aRecipe[13].RecipeLayerType[1].JobTableRight[0].SetTimeRamp := 0;
   aRecipe[13].RecipeLayerType[2].JobTableRight[0].SetTimeRamp := 0;
   aRecipe[14].RecipeLayerType[1].JobTableRight[0].SetTimeRamp := 0;
   aRecipe[14].RecipeLayerType[2].JobTableRight[0].SetTimeRamp := 0;
   aRecipe[15].RecipeLayerType[1].JobTableRight[0].SetTimeRamp := 0;
   aRecipe[15].RecipeLayerType[2].JobTableRight[0].SetTimeRamp := 0;
   aRecipe[16].RecipeLayerType[1].JobTableRight[0].SetTimeRamp := 0;
   aRecipe[16].RecipeLayerType[2].JobTableRight[0].SetTimeRamp := 0;
   aRecipe[17].RecipeLayerType[1].JobTableRight[0].SetTimeRamp := 0;
   aRecipe[17].RecipeLayerType[1].JobTableRight[1].SetTimeRamp := 2;
   aRecipe[17].RecipeLayerType[2].JobTableRight[0].SetTimeRamp := 0;
   aRecipe[18].RecipeLayerType[1].JobTableRight[0].SetTimeRamp := 0;
   aRecipe[18].RecipeLayerType[2].JobTableRight[0].SetTimeRamp := 0;
   aRecipe[19].RecipeLayerType[1].JobTableRight[0].SetTimeRamp := 0;
   aRecipe[19].RecipeLayerType[2].JobTableRight[0].SetTimeRamp := 0;
   aRecipe[20].RecipeLayerType[1].JobTableRight[0].SetTimeRamp := 0;
   aRecipe[20].RecipeLayerType[2].JobTableRight[0].SetTimeRamp := 0;
   aRecipe[21].RecipeLayerType[1].JobTableRight[0].SetTimeRamp := 0;
   aRecipe[21].RecipeLayerType[2].JobTableRight[0].SetTimeRamp := 0;
   aRecipe[22].RecipeLayerType[1].JobTableRight[0].SetTimeRamp := 0;
   aRecipe[22].RecipeLayerType[2].JobTableRight[0].SetTimeRamp := 0;
   aRecipe[23].RecipeLayerType[1].JobTableRight[0].SetTimeRamp := 0;
   aRecipe[23].RecipeLayerType[2].JobTableRight[0].SetTimeRamp := 0;
   aRecipe[1].RecipeLayerType[1].JobTableRight[0].SetSpeed := 0;
   aRecipe[1].RecipeLayerType[2].JobTableRight[0].SetSpeed := 0;
   aRecipe[2].RecipeLayerType[1].JobTableRight[0].SetSpeed := 0;
   aRecipe[2].RecipeLayerType[2].JobTableRight[0].SetSpeed := 0;
   aRecipe[3].RecipeLayerType[1].JobTableRight[0].SetSpeed := 0;
   aRecipe[3].RecipeLayerType[2].JobTableRight[0].SetSpeed := 0;
   aRecipe[4].RecipeLayerType[1].JobTableRight[0].SetSpeed := 0;
   aRecipe[4].RecipeLayerType[2].JobTableRight[0].SetSpeed := 0;
   aRecipe[5].RecipeLayerType[1].JobTableRight[0].SetSpeed := 0;
   aRecipe[5].RecipeLayerType[2].JobTableRight[0].SetSpeed := 0;
   aRecipe[6].RecipeLayerType[1].JobTableRight[0].SetSpeed := 0;
   aRecipe[6].RecipeLayerType[2].JobTableRight[0].SetSpeed := 0;
   aRecipe[7].RecipeLayerType[1].JobTableRight[0].SetSpeed := 0;
   aRecipe[7].RecipeLayerType[2].JobTableRight[0].SetSpeed := 0;
   aRecipe[8].RecipeLayerType[1].JobTableRight[0].SetSpeed := 0;
   aRecipe[8].RecipeLayerType[2].JobTableRight[0].SetSpeed := 0;
   aRecipe[9].RecipeLayerType[1].JobTableRight[0].SetSpeed := 0;
   aRecipe[9].RecipeLayerType[2].JobTableRight[0].SetSpeed := 0;
   aRecipe[10].RecipeLayerType[1].JobTableRight[0].SetSpeed := 0;
   aRecipe[10].RecipeLayerType[2].JobTableRight[0].SetSpeed := 0;
   aRecipe[11].RecipeLayerType[1].JobTableRight[0].SetSpeed := 0;
   aRecipe[11].RecipeLayerType[2].JobTableRight[0].SetSpeed := 0;
   aRecipe[12].RecipeLayerType[1].JobTableRight[0].SetSpeed := 0;
   aRecipe[12].RecipeLayerType[2].JobTableRight[0].SetSpeed := 0;
   aRecipe[13].RecipeLayerType[1].JobTableRight[0].SetSpeed := 0;
   aRecipe[13].RecipeLayerType[2].JobTableRight[0].SetSpeed := 0;
   aRecipe[14].RecipeLayerType[1].JobTableRight[0].SetSpeed := 0;
   aRecipe[14].RecipeLayerType[2].JobTableRight[0].SetSpeed := 0;
   aRecipe[15].RecipeLayerType[1].JobTableRight[0].SetSpeed := 0;
   aRecipe[15].RecipeLayerType[2].JobTableRight[0].SetSpeed := 0;
   aRecipe[16].RecipeLayerType[1].JobTableRight[0].SetSpeed := 0;
   aRecipe[16].RecipeLayerType[2].JobTableRight[0].SetSpeed := 0;
   aRecipe[17].RecipeLayerType[1].JobTableRight[0].SetSpeed := 0;
   aRecipe[17].RecipeLayerType[1].JobTableRight[1].SetSpeed := 4000;
   aRecipe[17].RecipeLayerType[2].JobTableRight[0].SetSpeed := 0;
   aRecipe[18].RecipeLayerType[1].JobTableRight[0].SetSpeed := 0;
   aRecipe[18].RecipeLayerType[2].JobTableRight[0].SetSpeed := 0;
   aRecipe[19].RecipeLayerType[1].JobTableRight[0].SetSpeed := 0;
   aRecipe[19].RecipeLayerType[2].JobTableRight[0].SetSpeed := 0;
   aRecipe[20].RecipeLayerType[1].JobTableRight[0].SetSpeed := 0;
   aRecipe[20].RecipeLayerType[2].JobTableRight[0].SetSpeed := 0;
   aRecipe[21].RecipeLayerType[1].JobTableRight[0].SetSpeed := 0;
   aRecipe[21].RecipeLayerType[2].JobTableRight[0].SetSpeed := 0;
   aRecipe[22].RecipeLayerType[1].JobTableRight[0].SetSpeed := 0;
   aRecipe[22].RecipeLayerType[2].JobTableRight[0].SetSpeed := 0;
   aRecipe[23].RecipeLayerType[1].JobTableRight[0].SetSpeed := 0;
   aRecipe[23].RecipeLayerType[2].JobTableRight[0].SetSpeed := 0;
   aRecipe[1].RecipeLayerType[1].JobTableRight[0].SetRobotSpeed := 0;
   aRecipe[1].RecipeLayerType[2].JobTableRight[0].SetRobotSpeed := 0;
   aRecipe[2].RecipeLayerType[1].JobTableRight[0].SetRobotSpeed := 0;
   aRecipe[2].RecipeLayerType[1].JobTableRight[1..2].SetRobotSpeed := 300;
   aRecipe[2].RecipeLayerType[2].JobTableRight[0].SetRobotSpeed := 0;
   aRecipe[2].RecipeLayerType[2].JobTableRight[1..2].SetRobotSpeed := 300;
   aRecipe[3].RecipeLayerType[1].JobTableRight[0].SetRobotSpeed := 0;
   aRecipe[3].RecipeLayerType[1].JobTableRight[1].SetRobotSpeed := 200;
   aRecipe[3].RecipeLayerType[1].JobTableRight[2].SetRobotSpeed := 300;
   aRecipe[3].RecipeLayerType[2].JobTableRight[0].SetRobotSpeed := 0;
   aRecipe[3].RecipeLayerType[2].JobTableRight[1].SetRobotSpeed := 300;
   aRecipe[4].RecipeLayerType[1].JobTableRight[0].SetRobotSpeed := 0;
   aRecipe[4].RecipeLayerType[2].JobTableRight[0].SetRobotSpeed := 0;
   aRecipe[5].RecipeLayerType[1].JobTableRight[0].SetRobotSpeed := 0;
   aRecipe[5].RecipeLayerType[2].JobTableRight[0].SetRobotSpeed := 0;
   aRecipe[6].RecipeLayerType[1].JobTableRight[0].SetRobotSpeed := 0;
   aRecipe[6].RecipeLayerType[2].JobTableRight[0].SetRobotSpeed := 0;
   aRecipe[7].RecipeLayerType[1].JobTableRight[0].SetRobotSpeed := 0;
   aRecipe[7].RecipeLayerType[2].JobTableRight[0].SetRobotSpeed := 0;
   aRecipe[8].RecipeLayerType[1].JobTableRight[0].SetRobotSpeed := 0;
   aRecipe[8].RecipeLayerType[2].JobTableRight[0].SetRobotSpeed := 0;
   aRecipe[9].RecipeLayerType[1].JobTableRight[0].SetRobotSpeed := 0;
   aRecipe[9].RecipeLayerType[2].JobTableRight[0].SetRobotSpeed := 0;
   aRecipe[10].RecipeLayerType[1].JobTableRight[0].SetRobotSpeed := 0;
   aRecipe[10].RecipeLayerType[2].JobTableRight[0].SetRobotSpeed := 0;
   aRecipe[11].RecipeLayerType[1].JobTableRight[0].SetRobotSpeed := 0;
   aRecipe[11].RecipeLayerType[2].JobTableRight[0].SetRobotSpeed := 0;
   aRecipe[12].RecipeLayerType[1].JobTableRight[0].SetRobotSpeed := 0;
   aRecipe[12].RecipeLayerType[2].JobTableRight[0].SetRobotSpeed := 0;
   aRecipe[13].RecipeLayerType[1].JobTableRight[0].SetRobotSpeed := 0;
   aRecipe[13].RecipeLayerType[2].JobTableRight[0].SetRobotSpeed := 0;
   aRecipe[14].RecipeLayerType[1].JobTableRight[0].SetRobotSpeed := 0;
   aRecipe[14].RecipeLayerType[2].JobTableRight[0].SetRobotSpeed := 0;
   aRecipe[15].RecipeLayerType[1].JobTableRight[0].SetRobotSpeed := 0;
   aRecipe[15].RecipeLayerType[2].JobTableRight[0].SetRobotSpeed := 0;
   aRecipe[16].RecipeLayerType[1].JobTableRight[0].SetRobotSpeed := 0;
   aRecipe[16].RecipeLayerType[2].JobTableRight[0].SetRobotSpeed := 0;
   aRecipe[17].RecipeLayerType[1].JobTableRight[0].SetRobotSpeed := 0;
   aRecipe[17].RecipeLayerType[1].JobTableRight[1].SetRobotSpeed := 150;
   aRecipe[17].RecipeLayerType[2].JobTableRight[0].SetRobotSpeed := 0;
   aRecipe[18].RecipeLayerType[1].JobTableRight[0].SetRobotSpeed := 0;
   aRecipe[18].RecipeLayerType[2].JobTableRight[0].SetRobotSpeed := 0;
   aRecipe[19].RecipeLayerType[1].JobTableRight[0].SetRobotSpeed := 0;
   aRecipe[19].RecipeLayerType[2].JobTableRight[0].SetRobotSpeed := 0;
   aRecipe[20].RecipeLayerType[1].JobTableRight[0].SetRobotSpeed := 0;
   aRecipe[20].RecipeLayerType[2].JobTableRight[0].SetRobotSpeed := 0;
   aRecipe[21].RecipeLayerType[1].JobTableRight[0].SetRobotSpeed := 0;
   aRecipe[21].RecipeLayerType[2].JobTableRight[0].SetRobotSpeed := 0;
   aRecipe[22].RecipeLayerType[1].JobTableRight[0].SetRobotSpeed := 0;
   aRecipe[22].RecipeLayerType[2].JobTableRight[0].SetRobotSpeed := 0;
   aRecipe[23].RecipeLayerType[1].JobTableRight[0].SetRobotSpeed := 0;
   aRecipe[23].RecipeLayerType[2].JobTableRight[0].SetRobotSpeed := 0;
   aRecipe[1].RecipeLayerType[1].JobTableRight[0].WornPaperDistance := 0;
   aRecipe[1].RecipeLayerType[2].JobTableRight[0].WornPaperDistance := 0;
   aRecipe[2].RecipeLayerType[1].JobTableRight[0].WornPaperDistance := 0;
   aRecipe[2].RecipeLayerType[1].JobTableRight[1].WornPaperDistance := 8;
   aRecipe[2].RecipeLayerType[1].JobTableRight[2].WornPaperDistance := 30;
   aRecipe[2].RecipeLayerType[2].JobTableRight[0].WornPaperDistance := 0;
   aRecipe[2].RecipeLayerType[2].JobTableRight[1..2].WornPaperDistance := 30;
   aRecipe[3].RecipeLayerType[1].JobTableRight[0].WornPaperDistance := 0;
   aRecipe[3].RecipeLayerType[1].JobTableRight[1..2].WornPaperDistance := 30;
   aRecipe[3].RecipeLayerType[2].JobTableRight[0].WornPaperDistance := 0;
   aRecipe[3].RecipeLayerType[2].JobTableRight[1].WornPaperDistance := 30;
   aRecipe[4].RecipeLayerType[1].JobTableRight[0].WornPaperDistance := 0;
   aRecipe[4].RecipeLayerType[2].JobTableRight[0].WornPaperDistance := 0;
   aRecipe[5].RecipeLayerType[1].JobTableRight[0].WornPaperDistance := 0;
   aRecipe[5].RecipeLayerType[2].JobTableRight[0].WornPaperDistance := 0;
   aRecipe[6].RecipeLayerType[1].JobTableRight[0].WornPaperDistance := 0;
   aRecipe[6].RecipeLayerType[2].JobTableRight[0].WornPaperDistance := 0;
   aRecipe[7].RecipeLayerType[1].JobTableRight[0].WornPaperDistance := 0;
   aRecipe[7].RecipeLayerType[2].JobTableRight[0].WornPaperDistance := 0;
   aRecipe[8].RecipeLayerType[1].JobTableRight[0].WornPaperDistance := 0;
   aRecipe[8].RecipeLayerType[2].JobTableRight[0].WornPaperDistance := 0;
   aRecipe[9].RecipeLayerType[1].JobTableRight[0].WornPaperDistance := 0;
   aRecipe[9].RecipeLayerType[2].JobTableRight[0].WornPaperDistance := 0;
   aRecipe[10].RecipeLayerType[1].JobTableRight[0].WornPaperDistance := 0;
   aRecipe[10].RecipeLayerType[2].JobTableRight[0].WornPaperDistance := 0;
   aRecipe[11].RecipeLayerType[1].JobTableRight[0].WornPaperDistance := 0;
   aRecipe[11].RecipeLayerType[2].JobTableRight[0].WornPaperDistance := 0;
   aRecipe[12].RecipeLayerType[1].JobTableRight[0].WornPaperDistance := 0;
   aRecipe[12].RecipeLayerType[2].JobTableRight[0].WornPaperDistance := 0;
   aRecipe[13].RecipeLayerType[1].JobTableRight[0].WornPaperDistance := 0;
   aRecipe[13].RecipeLayerType[2].JobTableRight[0].WornPaperDistance := 0;
   aRecipe[14].RecipeLayerType[1].JobTableRight[0].WornPaperDistance := 0;
   aRecipe[14].RecipeLayerType[2].JobTableRight[0].WornPaperDistance := 0;
   aRecipe[15].RecipeLayerType[1].JobTableRight[0].WornPaperDistance := 0;
   aRecipe[15].RecipeLayerType[2].JobTableRight[0].WornPaperDistance := 0;
   aRecipe[16].RecipeLayerType[1].JobTableRight[0].WornPaperDistance := 0;
   aRecipe[16].RecipeLayerType[2].JobTableRight[0].WornPaperDistance := 0;
   aRecipe[17].RecipeLayerType[1].JobTableRight[0].WornPaperDistance := 0;
   aRecipe[17].RecipeLayerType[2].JobTableRight[0].WornPaperDistance := 0;
   aRecipe[18].RecipeLayerType[1].JobTableRight[0].WornPaperDistance := 0;
   aRecipe[18].RecipeLayerType[2].JobTableRight[0].WornPaperDistance := 0;
   aRecipe[19].RecipeLayerType[1].JobTableRight[0].WornPaperDistance := 0;
   aRecipe[19].RecipeLayerType[2].JobTableRight[0].WornPaperDistance := 0;
   aRecipe[20].RecipeLayerType[1].JobTableRight[0].WornPaperDistance := 0;
   aRecipe[20].RecipeLayerType[2].JobTableRight[0].WornPaperDistance := 0;
   aRecipe[21].RecipeLayerType[1].JobTableRight[0].WornPaperDistance := 0;
   aRecipe[21].RecipeLayerType[2].JobTableRight[0].WornPaperDistance := 0;
   aRecipe[22].RecipeLayerType[1].JobTableRight[0].WornPaperDistance := 0;
   aRecipe[22].RecipeLayerType[2].JobTableRight[0].WornPaperDistance := 0;
   aRecipe[23].RecipeLayerType[1].JobTableRight[0].WornPaperDistance := 0;
   aRecipe[23].RecipeLayerType[2].JobTableRight[0].WornPaperDistance := 0;
   aRecipe[1].RecipeLayerType[1].JobTableRight[0].Gimball := 0;
   aRecipe[1].RecipeLayerType[2].JobTableRight[0].Gimball := 0;
   aRecipe[1].RecipeLayerType[2].JobTableRight[1].Gimball := 2;
   aRecipe[2].RecipeLayerType[1].JobTableRight[0].Gimball := 0;
   aRecipe[2].RecipeLayerType[2].JobTableRight[0].Gimball := 0;
   aRecipe[3].RecipeLayerType[1].JobTableRight[0].Gimball := 0;
   aRecipe[3].RecipeLayerType[2].JobTableRight[0].Gimball := 0;
   aRecipe[3].RecipeLayerType[2].JobTableRight[1].Gimball := 1;
   aRecipe[4].RecipeLayerType[1].JobTableRight[0].Gimball := 0;
   aRecipe[4].RecipeLayerType[2].JobTableRight[0].Gimball := 0;
   aRecipe[5].RecipeLayerType[1].JobTableRight[0].Gimball := 0;
   aRecipe[5].RecipeLayerType[2].JobTableRight[0].Gimball := 0;
   aRecipe[6].RecipeLayerType[1].JobTableRight[0].Gimball := 0;
   aRecipe[6].RecipeLayerType[2].JobTableRight[0].Gimball := 0;
   aRecipe[7].RecipeLayerType[1].JobTableRight[0].Gimball := 0;
   aRecipe[7].RecipeLayerType[2].JobTableRight[0].Gimball := 0;
   aRecipe[8].RecipeLayerType[1].JobTableRight[0].Gimball := 0;
   aRecipe[8].RecipeLayerType[2].JobTableRight[0].Gimball := 0;
   aRecipe[9].RecipeLayerType[1].JobTableRight[0].Gimball := 0;
   aRecipe[9].RecipeLayerType[2].JobTableRight[0].Gimball := 0;
   aRecipe[10].RecipeLayerType[1].JobTableRight[0].Gimball := 0;
   aRecipe[10].RecipeLayerType[2].JobTableRight[0].Gimball := 0;
   aRecipe[11].RecipeLayerType[1].JobTableRight[0].Gimball := 0;
   aRecipe[11].RecipeLayerType[2].JobTableRight[0].Gimball := 0;
   aRecipe[12].RecipeLayerType[1].JobTableRight[0].Gimball := 0;
   aRecipe[12].RecipeLayerType[2].JobTableRight[0].Gimball := 0;
   aRecipe[13].RecipeLayerType[1].JobTableRight[0].Gimball := 0;
   aRecipe[13].RecipeLayerType[2].JobTableRight[0].Gimball := 0;
   aRecipe[14].RecipeLayerType[1].JobTableRight[0].Gimball := 0;
   aRecipe[14].RecipeLayerType[2].JobTableRight[0].Gimball := 0;
   aRecipe[15].RecipeLayerType[1].JobTableRight[0].Gimball := 0;
   aRecipe[15].RecipeLayerType[2].JobTableRight[0].Gimball := 0;
   aRecipe[16].RecipeLayerType[1].JobTableRight[0].Gimball := 0;
   aRecipe[16].RecipeLayerType[2].JobTableRight[0].Gimball := 0;
   aRecipe[17].RecipeLayerType[1].JobTableRight[0].Gimball := 0;
   aRecipe[17].RecipeLayerType[1].JobTableRight[1].Gimball := 1;
   aRecipe[17].RecipeLayerType[2].JobTableRight[0].Gimball := 0;
   aRecipe[18].RecipeLayerType[1].JobTableRight[0].Gimball := 0;
   aRecipe[18].RecipeLayerType[2].JobTableRight[0].Gimball := 0;
   aRecipe[19].RecipeLayerType[1].JobTableRight[0].Gimball := 0;
   aRecipe[19].RecipeLayerType[2].JobTableRight[0].Gimball := 0;
   aRecipe[20].RecipeLayerType[1].JobTableRight[0].Gimball := 0;
   aRecipe[20].RecipeLayerType[2].JobTableRight[0].Gimball := 0;
   aRecipe[21].RecipeLayerType[1].JobTableRight[0].Gimball := 0;
   aRecipe[21].RecipeLayerType[2].JobTableRight[0].Gimball := 0;
   aRecipe[22].RecipeLayerType[1].JobTableRight[0].Gimball := 0;
   aRecipe[22].RecipeLayerType[2].JobTableRight[0].Gimball := 0;
   aRecipe[23].RecipeLayerType[1].JobTableRight[0].Gimball := 0;
   aRecipe[23].RecipeLayerType[2].JobTableRight[0].Gimball := 0;
   aRecipe[1].RecipeLayerType[2].JobTableRight[1].UnlockEccentric1 := TRUE;
   aRecipe[1].RecipeLayerType[2].JobTableRight[1].UnlockEccentric2 := TRUE;
   aRecipe[1].RecipeLayerType[2].JobTableRight[1].UnlockEccentric3 := TRUE;
END_DATA_BLOCK

DATA_BLOCK "DB_Fault"   // DB60
{ S7_Optimized_Access := 'TRUE'; DB_Accessible_From_OPC_UA := 'FALSE' }
// stored: AutoNumber false, DBAccessibleFromOPCUA false, DBAccessibleFromWebserver false, MemoryReserve 100
   VAR
      tonFaultAirPressureLeftRobot { ExternalAccessible := 'False'; ExternalVisible := 'False'; ExternalWritable := 'False'; S7_SetPoint := 'True'} : TON_TIME;
      tonFaultAirPressureRightRobot { ExternalAccessible := 'False'; ExternalVisible := 'False'; ExternalWritable := 'False'; S7_SetPoint := 'True'} : TON_TIME;
      tonFaultAirPressureVacuum { ExternalAccessible := 'False'; ExternalVisible := 'False'; ExternalWritable := 'False'; S7_SetPoint := 'True'} : TON_TIME;
      tonFaultVacuumPumpRunning { ExternalAccessible := 'False'; ExternalVisible := 'False'; ExternalWritable := 'False'; S7_SetPoint := 'True'} : TON_TIME;
   END_VAR
BEGIN
END_DATA_BLOCK

DATA_BLOCK "DB_ExportFlatCtrlRobot1"   // DB72
{ S7_Optimized_Access := 'TRUE' }
// stored: AutoNumber false, IsOnlyStoredInLoadMemory true, MemoryReserve 100
   VAR RETAIN
      FlatnessRecords { S7_SetPoint := 'True'} : Array[0..200] of "stFlatnessCtrlRecord";
   END_VAR
BEGIN
   FlatnessRecords[1].dtlDataTime := DTL#2025-07-23-18:30:25.845572084;
   FlatnessRecords[1].xFlatnessResult := TRUE;
   FlatnessRecords[1].uiStrokePositionDiskA := 237;
   FlatnessRecords[1].uiStrokePositionDiskB := 237;
   FlatnessRecords[1].uiStrokePositionDiskC := 240;
END_DATA_BLOCK

DATA_BLOCK "DB_ExportFlatCtrlRobot2"   // DB73
{ S7_Optimized_Access := 'TRUE' }
// stored: AutoNumber false, IsOnlyStoredInLoadMemory true, MemoryReserve 100
   VAR RETAIN
      FlatnessRecords { S7_SetPoint := 'True'} : Array[0..200] of "stFlatnessCtrlRecord";
   END_VAR
BEGIN
   FlatnessRecords[1].dtlDataTime := DTL#2025-07-23-18:25:23.687016057;
   FlatnessRecords[1].xFlatnessResult := TRUE;
   FlatnessRecords[1].uiStrokePositionDiskA := 239;
   FlatnessRecords[1].uiStrokePositionDiskB := 236;
   FlatnessRecords[1].uiStrokePositionDiskC := 237;
END_DATA_BLOCK

DATA_BLOCK "DB_ExportProdData"   // DB71
{ S7_Optimized_Access := 'TRUE' }
// stored: AutoNumber false, IsOnlyStoredInLoadMemory true, MemoryReserve 100
   VAR RETAIN
      aProdData { S7_SetPoint := 'True'} : Array[0..200] of "stProductionRecord";
   END_VAR
BEGIN
   aProdData[1..2].dDate := D#2025-07-29;
   aProdData[1].todTime := TOD#13:18:42.636;
   aProdData[2].todTime := TOD#11:56:55.157;
   aProdData[1..2].sRecipeName := 'Test Carbody Shell';
   aProdData[1..2].usiProgNumber := 101;
   aProdData[1..2].sRecipeLayerTypeName := 'Putty Layer';
   aProdData[1..2].usiLayerTypeNumber := 1;
   aProdData[1].uiCbsNumber := 45;
   aProdData[2].uiCbsNumber := 46;
   aProdData[1].uiPaperUsed := 6;
   aProdData[1].tCycleTime := TOD#00:06:08.019;
   aProdData[2].tCycleTime := TOD#01:12:43.602;
END_DATA_BLOCK

DATA_BLOCK "DB_FlatnessCtrlRecords"   // DB77
{ S7_Optimized_Access := 'TRUE'; DB_Accessible_From_OPC_UA := 'FALSE' }
// stored: AutoNumber false, DBAccessibleFromOPCUA false, DBAccessibleFromWebserver false, MemoryReserve 100
   VAR RETAIN
      LeftRobot { ExternalWritable := 'False'} : Struct
         uiNumberOfRecods : UInt;
         FlatnessRecords : Array[0..200] of "stFlatnessCtrlRecord";
      END_STRUCT;
      RightRobot { ExternalWritable := 'False'} : Struct
         uiNumberOfRecods : UInt;
         FlatnessRecords : Array[0..200] of "stFlatnessCtrlRecord";
      END_STRUCT;
   END_VAR
BEGIN
END_DATA_BLOCK

DATA_BLOCK "DB_ProductionRecords"   // DB76
{ S7_Optimized_Access := 'TRUE'; DB_Accessible_From_OPC_UA := 'FALSE' }
// stored: AutoNumber false, DBAccessibleFromOPCUA false, DBAccessibleFromWebserver false, MemoryReserve 100
   VAR RETAIN
      uiNumberOfRecords { ExternalWritable := 'False'} : UInt;
      aProdData { ExternalWritable := 'False'} : Array[0..200] of "stProductionRecord";
   END_VAR
BEGIN
END_DATA_BLOCK

